# B&R Automation Studio project pneutrunk_plc
Automation Studio 4.9

## Configuration Config1

### Task classes (Cpu.sw)
```
Cyclic#1 (cycle 2000 us, tolerance 2000 us):
  Server <- Source.UDP.Server.prg
  Client <- Source.UDP.Client.prg
  Receiver <- (binary)
  Sender <- (binary)
Cyclic#2 (cycle 12000 us, tolerance 12000 us):
  Receiver1 <- Source.RS485.Receiver.prg
  test_input <- test_input.prg (AdditionalIncludeDirectories=\Logical\MATLAB_includes\R2023a\, BuildOptions=-lm -DMODEL=simulink_2_plc -DNUMST=2 -DNCSTATES=0 -DHAVESTDIO -DRT -DUSE_RTMODEL -DEXT_MODE -DEXTMODE_STATIC -DEXTMODE_STATIC_SIZE=1000000 -DON_TARGET_WAIT_FOR_START=0 -DCLASSIC_INTERFACE=1 -DALLOCATIONFCN=0 -DTID01EQ=1 -DMAT_FILE=0 -DONESTEPFCN=0 -DTERMFCN=1 -DMULTI_INSTANCE_CODE=0 -DINTEGER_CODE=0 -DMT=0 )
Cyclic#3 (cycle 16000 us, tolerance 16000 us):
  Sender1 <- Source.RS485.Sender.prg
  solo_reg <- solo_reg.prg (AdditionalIncludeDirectories=\Logical\MATLAB_includes\R2023a\, BuildOptions=-lm -DMODEL=pneutr2_reg_FF_stiff -DNUMST=1 -DNCSTATES=0 -DHAVESTDIO -DRT -DUSE_RTMODEL -DCLASSIC_INTERFACE=1 -DALLOCATIONFCN=0 -DTID01EQ=0 -DMAT_FILE=0 -DONESTEPFCN=0 -DTERMFCN=1 -DMULTI_INSTANCE_CODE=0 -DINTEGER_CODE=0 -DMT=0 )
Cyclic#4 (cycle 24000 us, tolerance 96000 us):
  Controller <- Source.Controller.prg
  Identifika <- Source.Identifikacia.prg [disabled]
  meranie <- meranie.prg [disabled] (AdditionalIncludeDirectories=\Logical\MATLAB_includes\R2022b\, BuildOptions=-lm -DMODEL=pneutrunkMeranie -DNUMST=1 -DNCSTATES=0 -DHAVESTDIO -DRT -DUSE_RTMODEL -DEXT_MODE -DEXTMODE_STATIC -DEXTMODE_STATIC_SIZE=1000000 -DON_TARGET_WAIT_FOR_START=0 -DCLASSIC_INTERFACE=1 -DALLOCATIONFCN=0 -DTID01EQ=0 -DMAT_FILE=0 -DONESTEPFCN=0 -DTERMFCN=1 -DMULTI_INSTANCE_CODE=0 -DINTEGER_CODE=0 -DMT=0 )
  Testing <- Source.Testing.prg [disabled]
  Program <- Source.Program.prg [disabled]
DataObjects: Acp10sys
Binaries: FWRules, TCData, udbdef, asfw, User, iomap, sysconf, arconfig, ashwd, Role, ashwac, Acp10map, acp10cfg
Libraries: runtime, AsUDP, asstring, standard, sys_lib, brsystem, dvframe, AsTCP, AsArLog, regulatory, asieccon, astime, powerlnk, fileio
```

### Hardware
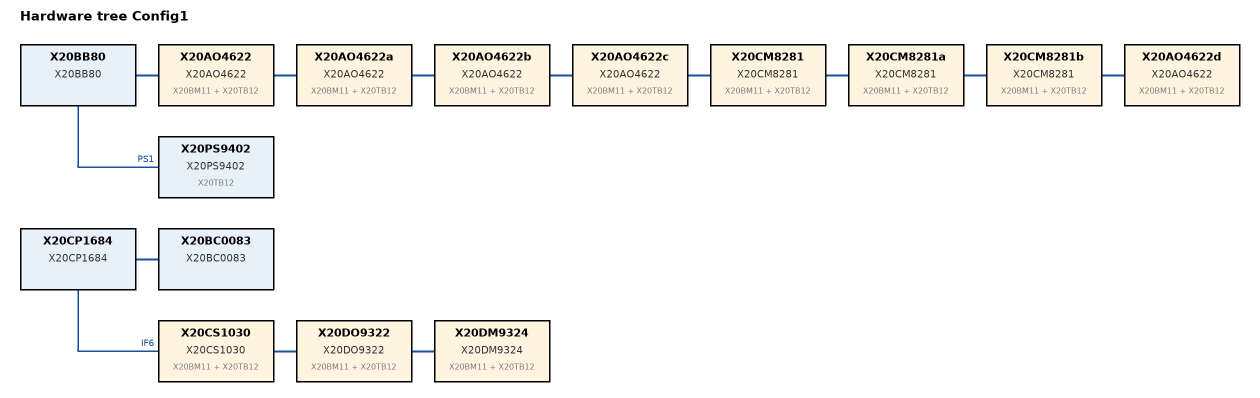
```
X20AO4622 : X20AO4622 v1.3.0.0  [SS1 -> X20TB12a.SS; SL -> X20BM11.SL1]
X20AO4622a : X20AO4622 v1.3.0.0  [SS1 -> X20TB12b.SS; SL -> X20BM11a.SL1]
X20AO4622b : X20AO4622 v1.3.0.0  [SS1 -> X20TB12c.SS; SL -> X20BM11b.SL1]
X20AO4622c : X20AO4622 v1.3.0.0  [SS1 -> X20TB12d.SS; SL -> X20BM11c.SL1]
X20AO4622d : X20AO4622 v1.3.0.0  [SS1 -> X20TB12i.SS; SL -> X20BM11h.SL1]
X20BB80 : X20BB80 v1.1.0.0
X20BC0083 : X20BC0083 v2.14.0.0  [PLK1 -> X20CP1684.IF3 (NodeNumber=1) [Cable Type=PowerlinkCable, Length=10, Version=1.0.0.3]; SL -> X20BB80.SL1]
X20BM11 : X20BM11 v1.1.0.0  [X2X1 -> X20BB80.IF1]
X20BM11a : X20BM11 v1.1.0.0  [X2X1 -> X20BM11.X2X2]
X20BM11b : X20BM11 v1.1.0.0  [X2X1 -> X20BM11a.X2X2]
X20BM11c : X20BM11 v1.1.0.0  [X2X1 -> X20BM11b.X2X2]
X20BM11d : X20BM11 v1.1.0.0  [X2X1 -> X20BM11c.X2X2]
X20BM11e : X20BM11 v1.1.0.0  [X2X1 -> X20BM11d.X2X2]
X20BM11f : X20BM11 v1.1.0.0  [X2X1 -> X20BM11e.X2X2]
X20BM11g : X20BM11 v1.1.0.0  [X2X1 -> X20CP1684.IF6]
X20BM11h : X20BM11 v1.1.0.0  [X2X1 -> X20BM11f.X2X2]
X20BM11i : X20BM11 v1.1.0.0  [X2X1 -> X20BM11g.X2X2]
X20BM11j : X20BM11 v1.1.0.0  [X2X1 -> X20BM11i.X2X2]
X20CM8281 : X20CM8281 v1.4.0.0  [SS1 -> X20TB12e.SS; SL -> X20BM11d.SL1]
X20CM8281a : X20CM8281 v1.4.0.0  [SS1 -> X20TB12f.SS; SL -> X20BM11e.SL1]
X20CM8281b : X20CM8281 v1.4.0.0  [SS1 -> X20TB12g.SS; SL -> X20BM11f.SL1]
X20CP1684 : X20CP1684 v1.5.0.0
  Connector IF2:
    ActivateDevice = 1
    ActivateSnmp = 2
  ConfigurationID = pneutrunk_Config1
  TimerDeviceType = EPLX2X
  TimerDevice = X20CP1684.IF3
  IdleTaskClass = 4
  TaskClassIdleTime = 2000
  Cyclic1Duration = 2000
  Cyclic1Tolerance = 2000
  Cyclic2Duration = 12000
  Cyclic2Tolerance = 12000
  Cyclic3Duration = 16000
  Cyclic3Tolerance = 16000
  Cyclic4Duration = 24000
  Cyclic4Tolerance = 96000
  Cyclic5Duration = 50000
  Cyclic5Tolerance = 50000
  FileDevice1
  FileDeviceName1 = USER
  FileDevicePath1 = USER_PATH
  ActivateDns = 1
  DnsDefaultDomain = br-automation.co.at
  ActivateOpcUa = 1
  OpcUa_Security_AdminRole = Administrators
  OpcUaInformationModels_PV_Version = 1
X20CS1030 : X20CS1030 v1.8.0.0  [SS1 -> X20TB12h.SS; SL -> X20BM11g.SL1]
  Connector IF1:
    Baudrate = 38400
    Parity = N
    DeviceType = RS485
  FunctionModel = StreamCyc1xRS4xx
X20DM9324 : X20DM9324 v1.2.0.0  [SS1 -> X20TB12k.SS; SL -> X20BM11j.SL1]
X20DO9322 : X20DO9322 v1.5.0.0  [SS1 -> X20TB12j.SS; SL -> X20BM11i.SL1]
X20PS9402 : X20PS9402 v1.2.0.0  [SS1 -> X20TB12.SS; PS -> X20BB80.PS1]
X20TB12 : X20TB12 v1.0.0.0
X20TB12a : X20TB12 v1.0.0.0
X20TB12b : X20TB12 v1.0.0.0
X20TB12c : X20TB12 v1.0.0.0
X20TB12d : X20TB12 v1.0.0.0
X20TB12e : X20TB12 v1.0.0.0
X20TB12f : X20TB12 v1.0.0.0
X20TB12g : X20TB12 v1.0.0.0
X20TB12h : X20TB12 v1.0.0.0
X20TB12i : X20TB12 v1.0.0.0
X20TB12j : X20TB12 v1.0.0.0
X20TB12k : X20TB12 v1.0.0.0
```

### IoMap.iom - X20CP1684/IoMap.iom
```iecst
VAR_CONFIG
	::modul.tlak2[5] AT %QW."X20CM8281".AnalogOutput01;
	::modul.tlak3[5] AT %QW."X20CM8281a".AnalogOutput01;
	::modul.tlak1[0] AT %QW."X20AO4622".AnalogOutput01;
	::modul.tlak2[0] AT %QW."X20AO4622".AnalogOutput02;
	::modul.tlak3[0] AT %QW."X20AO4622".AnalogOutput03;
	::modul.tlak1[1] AT %QW."X20AO4622".AnalogOutput04;
	::modul.tlak2[1] AT %QW."X20AO4622a".AnalogOutput01;
	::modul.tlak3[1] AT %QW."X20AO4622a".AnalogOutput02;
	::modul.tlak1[2] AT %QW."X20AO4622a".AnalogOutput03;
	::modul.tlak2[2] AT %QW."X20AO4622a".AnalogOutput04;
	::modul.tlak3[2] AT %QW."X20AO4622b".AnalogOutput01;
	::modul.tlak1[3] AT %QW."X20AO4622b".AnalogOutput02;
	::modul.tlak2[3] AT %QW."X20AO4622b".AnalogOutput03;
	::modul.tlak3[3] AT %QW."X20AO4622b".AnalogOutput04;
	::modul.tlak1[4] AT %QW."X20AO4622c".AnalogOutput01;
	::modul.tlak2[4] AT %QW."X20AO4622c".AnalogOutput02;
	::modul.tlak3[4] AT %QW."X20AO4622c".AnalogOutput03;
	::modul.tlak1[5] AT %QW."X20AO4622c".AnalogOutput04;
	::modul.tlakLinear AT %QW."X20CM8281b".AnalogOutput01;
	::Controller:modull.efektor AT %QX."X20CM8281".DigitalOutput01;
	::modul.tlak2[6] AT %QW."X20AO4622d".AnalogOutput01;
	::modul.tlak3[6] AT %QW."X20AO4622d".AnalogOutput02;
	::modul.tlak1[6] AT %QW."X20AO4622d".AnalogOutput03;
	::zasobnik.ball AT %QX."X20DO9322".DigitalOutput12;
	::zasobnik.ball_piston_sjf AT %QX."X20DO9322".DigitalOutput11;
	::zasobnik.ball_piston AT %QX."X20DO9322".DigitalOutput10;
	::zasobnik.levitovanie AT %QX."X20DO9322".DigitalOutput09;
	::buttons.stropCervenaLED AT %QX."X20DO9322".DigitalOutput08;
	::buttons.startLED AT %QX."X20DO9322".DigitalOutput06;
	::buttons.stopLED AT %QX."X20DO9322".DigitalOutput07;
	::buttons.stropBielaLED AT %QX."X20DO9322".DigitalOutput05;
	::buttons.startButton AT %IX."X20DM9324".DigitalInput01;
	::buttons.stop AT %IX."X20DM9324".DigitalInput02;
	::buttons.centralStop AT %IX."X20DM9324".DigitalInput04;
END_VAR
```

## Logical view

### Global.typ - Global data types
```iecst
TYPE
	tlacidla : 	STRUCT
		start : BOOL;
		ros : BOOL;
		stopLED : BOOL;
		stop : BOOL;
		startLED : BOOL;
		startButton : BOOL;
		centralStop : BOOL;
		stropBielaLED : BOOL;
		stropCervenaLED : BOOL;
		klucik : BOOL;
	END_STRUCT;
	automatic : 	STRUCT
		y_desired : ARRAY[0..6]OF INT := [7(0)];
		x_desired : ARRAY[0..6]OF INT := [7(0)];
		linear : INT;
		ball_up : BOOL;
		casovac : BOOL;
		effector : BOOL;
		casovac_uchopenie : BOOL;
		ball_piston : BOOL;
		novyCyklus : TIME := T#1s;
		novyCyklusStart : BOOL;
		trajectoryStart2 : BOOL;
		trajectoryTime2 : TIME := T#6s;
		automatic : BOOL;
		holdPosition : BOOL;
		cas : INT;
		box : INT;
		step_color : INT;
		popcorn : BOOL;
		testFarba : INT;
		loptickyVzasobniku : BOOL := TRUE;
		x_desired_previous : ARRAY[0..6]OF INT;
		y_desired_previous : ARRAY[0..6]OF INT;
		I_konstanta : ARRAY[0..6]OF INT;
		levitacia : BOOL;
	END_STRUCT;
	podavac : 	STRUCT
		levitovanie : BOOL;
		ball_piston_sjf : BOOL;
		ball : BOOL;
		ball_piston : BOOL;
	END_STRUCT;
	identifikacia : 	STRUCT
		p3 : REAL;
		p2 : REAL;
		p1 : REAL;
		vzorka : USINT;
		uhol2 : ARRAY[0..9]OF INT;
		uhol2Priemer : INT;
		uhol1Priemer : INT;
		uhol1 : ARRAY[0..9]OF INT;
		uhol2Stabilny : BOOL;
		uhol1Stabilny : BOOL;
		uhol2Ref : INT;
		uhol1Ref : INT;
		krok : USINT;
		p2Mem : REAL;
		p1Mem : REAL;
		tonStart : BOOL;
		pocetOverenie : USINT := 10;
		spustit : BOOL;
		p3Koniec : BOOL;
		p2Koniec : BOOL;
		p1Koniec : BOOL;
		p3Mem : REAL;
		results : INT;
		switchs : BOOL;
		inkrement : REAL;
		hornyTlak : REAL;
	END_STRUCT;
	packetRS485 : 	STRUCT
		packet : ARRAY[0..9]OF BYTE;
		sendPacketLED : ARRAY[0..5]OF BYTE;
		sendPacketSnimace : ARRAY[0..5]OF BYTE;
		sendPacketFinal : ARRAY[0..5]OF BYTE;
		id : USINT;
	END_STRUCT;
	packetUDP : 	STRUCT
		qLength : INT;
		c : INT;
		q : INT;
		qFull : STRING[80];
		comma : INT;
		qString : ARRAY[0..14]OF STRING[6];
		qDesired : ARRAY[0..14]OF REAL;
		color : INT;
		step : INT;
	END_STRUCT;
	tlaky : 	STRUCT
		tlak3 : USINT;
		tlak2 : USINT;
		tlak1 : USINT;
	END_STRUCT;
	moduly : 	STRUCT
		uhol2 : ARRAY[0..6]OF INT := [7(0)];
		uhol1 : ARRAY[0..6]OF INT := [7(0)];
		koncak : ARRAY[0..6]OF BOOL;
		led : ARRAY[0..6]OF BOOL;
		uholINT2 : INT;
		uholINT1 : INT;
		tlak1 : ARRAY[0..6]OF INT;
		tlak2 : ARRAY[0..6]OF INT;
		tlak3 : ARRAY[0..6]OF INT;
		tlakLinear : INT;
		uhol_XminusRef : ARRAY[0..6]OF REAL; (*uhol ktory posiela PLC do PC po odpocitani odchylky naklonenia realneho robota*)
		uhol_YminusRef : ARRAY[0..6]OF REAL; (*uhol ktory posiela PLC do PC po odpocitani odchylky naklonenia realneho robota*)
		linearReal : REAL;
		naraz : ARRAY[0..7]OF BOOL;
		narazAktivny : BOOL;
	END_STRUCT;
END_TYPE
```

### Global.var - Global variables
```iecst
VAR
	hranica_upravy_traj : REAL := 2;
	Yellow_tab_ID7 : REAL;
	zasobnik : podavac;
	Yellow_tab_ID6 : REAL;
	I_ON : BOOL;
	Yellow_tab_ID5 : REAL;
	step : INT;
	Yellow_tab_ID4 : REAL;
	Yellow_tab_ID3 : REAL;
	Yellow_tab_ID2 : REAL;
	automatika : automatic;
	Yellow_tab_ID1 : REAL;
	u2 : INT;
	u1 : INT;
	stiffness_ff : REAL;
	result : INT;
	RESET_ID7 : REAL;
	RESET_ID6 : REAL;
	RESET_ID5 : REAL;
	RESET_ID4 : REAL;
	RESET_ID3 : REAL;
	RESET_ID2 : REAL;
	RESET_ID1 : REAL;
	ref_linearny_posun : REAL;
	ref_alfa_y_ID7 : REAL;
	ref_alfa_y_ID6 : REAL;
	ref_alfa_y_ID5 : REAL;
	ref_alfa_y_ID4 : REAL;
	ref_alfa_y_ID3 : REAL;
	ref_alfa_y_ID2 : REAL;
	ref_alfa_y_ID1 : REAL;
	ref_alfa_x_ID7 : REAL;
	ref_alfa_x_ID6 : REAL;
	ref_alfa_x_ID5 : REAL;
	ref_alfa_x_ID4 : REAL;
	ref_alfa_x_ID3 : REAL;
	ref_alfa_x_ID2 : REAL;
	ref_alfa_x_ID1 : REAL;
	q_real : ARRAY[0..12] OF REAL := [0.55,12.58,12.23,7.85,1.23,15.36,17.85,12.05,3.85,3.6,-12.52,10.65,31.28];
	q_desired : ARRAY[0..12] OF REAL;
	pripustna_odchylka_naklonenia : REAL := 0.25;
	poradie_ID7 : REAL;
	poradie_ID6 : REAL;
	poradie_ID5 : REAL;
	poradie_ID4 : REAL;
	poradie_ID3 : REAL;
	poradie_ID2 : REAL;
	poradie_ID1 : REAL;
	packetPos : packetUDP;
	packet485 : packetRS485;
	p3 : REAL;
	p2 : REAL;
	p1 : REAL;
	modul : moduly;
	meranie : identifikacia;
	lin_pressure : REAL;
	I_konstanta_ID7 : REAL;
	I_konstanta_ID6 : REAL;
	I_konstanta_ID5 : REAL;
	I_konstanta_ID4 : REAL;
	I_konstanta_ID3 : REAL;
	I_konstanta_ID2 : REAL;
	cos_test_hodnota2 : REAL;
	cos_test_hodnota1 : REAL;
	I_konstanta_ID1 : REAL;
	Green_tab_ID7 : REAL;
	Green_tab_ID6 : REAL;
	trajectoryStart : BOOL;
	Green_tab_ID5 : REAL;
	Green_tab_ID4 : REAL;
	uhly : experimentyUhly;
	Green_tab_ID3 : REAL;
	Green_tab_ID2 : REAL;
	Green_tab_ID1 : REAL;
	step_color : INT;
	global_step_udp : INT;
	global_step : INT;
	datagramLength : INT;
	centralStop : BOOL;
	cas_trajektorie : REAL := 100;
	Blue_tab_ID7 : REAL;
	Blue_tab_ID6 : REAL;
	Blue_tab_ID5 : REAL;
	buttons : tlacidla;
	Blue_tab_ID4 : REAL;
	Blue_tab_ID3 : REAL;
	Blue_tab_ID2 : REAL;
	Blue_tab_ID1 : REAL;
	act_alfa_y_ID7 : REAL;
	act_alfa_y_ID6 : REAL;
	act_alfa_y_ID5 : REAL;
	step_repeatability : INT;
	act_alfa_y_ID4 : REAL;
	act_alfa_y_ID3 : REAL;
	act_alfa_y_ID2 : REAL;
	act_alfa_y_ID1 : REAL;
	act_alfa_x_ID7 : REAL;
	act_alfa_x_ID6 : REAL;
	act_alfa_x_ID5 : REAL;
	act_alfa_x_ID4 : REAL;
	act_alfa_x_ID3 : REAL;
	act_alfa_x_ID2 : REAL;
	act_alfa_x_ID1 : REAL;
END_VAR
```

### Package Logical/Libraries - Global libraries

### Program Logical/Libraries/regulatory

#### multiword_types.h
```c
/*
 * multiword_types.h
 *
 * Academic License - for use in teaching, academic research, and meeting
 * course requirements at degree granting institutions only.  Not for
 * government, commercial, or other organizational use.
 *
 * Code generation for model "reg_FF_PI_pl_regr_stiff".
 *
 * Model version              : 1.154
 * Simulink Coder version : 9.6 (R2021b) 14-May-2021
 * C source code generated on : Mon Jun 26 09:10:26 2023
 *
 * Target selection: bur_grt.tlc
 * Note: GRT includes extra infrastructure and instrumentation for prototyping
 * Embedded hardware selection: Intel->x86/Pentium
 * Code generation objectives: Unspecified
 * Validation result: Not run
 */

#ifndef MULTIWORD_TYPES_H
#define MULTIWORD_TYPES_H
#include "rtwtypes.h"

/*
 * MultiWord supporting definitions
 */
typedef long int long_T;

/*
 * MultiWord types
 */
typedef struct {
  uint32_T chunks[2];
} int64m_T;

typedef struct {
  int64m_T re;
  int64m_T im;
} cint64m_T;

typedef struct {
  uint32_T chunks[2];
} uint64m_T;

typedef struct {
  uint64m_T re;
  uint64m_T im;
} cuint64m_T;

typedef struct {
  uint32_T chunks[3];
} int96m_T;

typedef struct {
  int96m_T re;
  int96m_T im;
} cint96m_T;

typedef struct {
  uint32_T chunks[3];
} uint96m_T;

typedef struct {
  uint96m_T re;
  uint96m_T im;
} cuint96m_T;

typedef struct {
  uint32_T chunks[4];
} int128m_T;

typedef struct {
  int128m_T re;
  int128m_T im;
} cint128m_T;

typedef struct {
  uint32_T chunks[4];
} uint128m_T;

typedef struct {
  uint128m_T re;
  uint128m_T im;
} cuint128m_T;

typedef struct {
  uint32_T chunks[5];
} int160m_T;

typedef struct {
  int160m_T re;
  int160m_T im;
} cint160m_T;

typedef struct {
  uint32_T chunks[5];
} uint160m_T;

typedef struct {
  uint160m_T re;
  uint160m_T im;
} cuint160m_T;

typedef struct {
  uint32_T chunks[6];
} int192m_T;

typedef struct {
  int192m_T re;
  int192m_T im;
} cint192m_T;

typedef struct {
  uint32_T chunks[6];
} uint192m_T;

typedef struct {
  uint192m_T re;
  uint192m_T im;
} cuint192m_T;

typedef struct {
  uint32_T chunks[7];
} int224m_T;

typedef struct {
  int224m_T re;
  int224m_T im;
} cint224m_T;

typedef struct {
  uint32_T chunks[7];
} uint224m_T;

typedef struct {
  uint224m_T re;
  uint224m_T im;
} cuint224m_T;

typedef struct {
  uint32_T chunks[8];
} int256m_T;

typedef struct {
  int256m_T re;
  int256m_T im;
} cint256m_T;

typedef struct {
  uint32_T chunks[8];
} uint256m_T;

typedef struct {
  uint256m_T re;
  uint256m_T im;
} cuint256m_T;

typedef struct {
  uint32_T chunks[9];
} int288m_T;

typedef struct {
  int288m_T re;
  int288m_T im;
} cint288m_T;

typedef struct {
  uint32_T chunks[9];
} uint288m_T;

typedef struct {
  uint288m_T re;
  uint288m_T im;
} cuint288m_T;

typedef struct {
  uint32_T chunks[10];
} int320m_T;

typedef struct {
  int320m_T re;
  int320m_T im;
} cint320m_T;

typedef struct {
  uint32_T chunks[10];
} uint320m_T;

typedef struct {
  uint320m_T re;
  uint320m_T im;
} cuint320m_T;

typedef struct {
  uint32_T chunks[11];
} int352m_T;

typedef struct {
  int352m_T re;
  int352m_T im;
} cint352m_T;

typedef struct {
  uint32_T chunks[11];
} uint352m_T;

typedef struct {
  uint352m_T re;
  uint352m_T im;
} cuint352m_T;

typedef struct {
  uint32_T chunks[12];
} int384m_T;

typedef struct {
  int384m_T re;
  int384m_T im;
} cint384m_T;

typedef struct {
  uint32_T chunks[12];
} uint384m_T;

typedef struct {
  uint384m_T re;
  uint384m_T im;
} cuint384m_T;

typedef struct {
  uint32_T chunks[13];
} int416m_T;

typedef struct {
  int416m_T re;
  int416m_T im;
} cint416m_T;

typedef struct {
  uint32_T chunks[13];
} uint416m_T;

typedef struct {
  uint416m_T re;
  uint416m_T im;
} cuint416m_T;

typedef struct {
  uint32_T chunks[14];
} int448m_T;

typedef struct {
  int448m_T re;
  int448m_T im;
} cint448m_T;

typedef struct {
  uint32_T chunks[14];
} uint448m_T;

typedef struct {
  uint448m_T re;
  uint448m_T im;
} cuint448m_T;

typedef struct {
  uint32_T chunks[15];
} int480m_T;

typedef struct {
  int480m_T re;
  int480m_T im;
} cint480m_T;

typedef struct {
  uint32_T chunks[15];
} uint480m_T;

typedef struct {
  uint480m_T re;
  uint480m_T im;
} cuint480m_T;

typedef struct {
  uint32_T chunks[16];
} int512m_T;

typedef struct {
  int512m_T re;
  int512m_T im;
} cint512m_T;

typedef struct {
  uint32_T chunks[16];
} uint512m_T;

typedef struct {
  uint512m_T re;
  uint512m_T im;
} cuint512m_T;

typedef struct {
  uint32_T chunks[17];
} int544m_T;

typedef struct {
  int544m_T re;
  int544m_T im;
} cint544m_T;

typedef struct {
  uint32_T chunks[17];
} uint544m_T;

typedef struct {
  uint544m_T re;
  uint544m_T im;
} cuint544m_T;

typedef struct {
  uint32_T chunks[18];
} int576m_T;

typedef struct {
  int576m_T re;
  int576m_T im;
} cint576m_T;

typedef struct {
  uint32_T chunks[18];
} uint576m_T;

typedef struct {
  uint576m_T re;
  uint576m_T im;
} cuint576m_T;

typedef struct {
  uint32_T chunks[19];
} int608m_T;

typedef struct {
  int608m_T re;
  int608m_T im;
} cint608m_T;

typedef struct {
  uint32_T chunks[19];
} uint608m_T;

typedef struct {
  uint608m_T re;
  uint608m_T im;
} cuint608m_T;

typedef struct {
  uint32_T chunks[20];
} int640m_T;

typedef struct {
  int640m_T re;
  int640m_T im;
} cint640m_T;

typedef struct {
  uint32_T chunks[20];
} uint640m_T;

typedef struct {
  uint640m_T re;
  uint640m_T im;
} cuint640m_T;

typedef struct {
  uint32_T chunks[21];
} int672m_T;

typedef struct {
  int672m_T re;
  int672m_T im;
} cint672m_T;

typedef struct {
  uint32_T chunks[21];
} uint672m_T;

typedef struct {
  uint672m_T re;
  uint672m_T im;
} cuint672m_T;

typedef struct {
  uint32_T chunks[22];
} int704m_T;

typedef struct {
  int704m_T re;
  int704m_T im;
} cint704m_T;

typedef struct {
  uint32_T chunks[22];
} uint704m_T;

typedef struct {
  uint704m_T re;
  uint704m_T im;
} cuint704m_T;

typedef struct {
  uint32_T chunks[23];
} int736m_T;

typedef struct {
  int736m_T re;
  int736m_T im;
} cint736m_T;

typedef struct {
  uint32_T chunks[23];
} uint736m_T;

typedef struct {
  uint736m_T re;
  uint736m_T im;
} cuint736m_T;

typedef struct {
  uint32_T chunks[24];
} int768m_T;

typedef struct {
  int768m_T re;
  int768m_T im;
} cint768m_T;

typedef struct {
  uint32_T chunks[24];
} uint768m_T;

typedef struct {
  uint768m_T re;
  uint768m_T im;
} cuint768m_T;

typedef struct {
  uint32_T chunks[25];
} int800m_T;

typedef struct {
  int800m_T re;
  int800m_T im;
} cint800m_T;

typedef struct {
  uint32_T chunks[25];
} uint800m_T;

typedef struct {
  uint800m_T re;
  uint800m_T im;
} cuint800m_T;

typedef struct {
  uint32_T chunks[26];
} int832m_T;

typedef struct {
  int832m_T re;
  int832m_T im;
} cint832m_T;

typedef struct {
  uint32_T chunks[26];
} uint832m_T;

typedef struct {
  uint832m_T re;
  uint832m_T im;
} cuint832m_T;

typedef struct {
  uint32_T chunks[27];
} int864m_T;

typedef struct {
  int864m_T re;
  int864m_T im;
} cint864m_T;

typedef struct {
  uint32_T chunks[27];
} uint864m_T;

typedef struct {
  uint864m_T re;
  uint864m_T im;
} cuint864m_T;

typedef struct {
  uint32_T chunks[28];
} int896m_T;

typedef struct {
  int896m_T re;
  int896m_T im;
} cint896m_T;

typedef struct {
  uint32_T chunks[28];
} uint896m_T;

typedef struct {
  uint896m_T re;
  uint896m_T im;
} cuint896m_T;

typedef struct {
  uint32_T chunks[29];
} int928m_T;

typedef struct {
  int928m_T re;
  int928m_T im;
} cint928m_T;

typedef struct {
  uint32_T chunks[29];
} uint928m_T;

typedef struct {
  uint928m_T re;
  uint928m_T im;
} cuint928m_T;

typedef struct {
  uint32_T chunks[30];
} int960m_T;

typedef struct {
  int960m_T re;
  int960m_T im;
} cint960m_T;

typedef struct {
  uint32_T chunks[30];
} uint960m_T;

typedef struct {
  uint960m_T re;
  uint960m_T im;
} cuint960m_T;

typedef struct {
  uint32_T chunks[31];
} int992m_T;

typedef struct {
  int992m_T re;
  int992m_T im;
} cint992m_T;

typedef struct {
  uint32_T chunks[31];
} uint992m_T;

typedef struct {
  uint992m_T re;
  uint992m_T im;
} cuint992m_T;

typedef struct {
  uint32_T chunks[32];
} int1024m_T;

typedef struct {
  int1024m_T re;
  int1024m_T im;
} cint1024m_T;

typedef struct {
  uint32_T chunks[32];
} uint1024m_T;

typedef struct {
  uint1024m_T re;
  uint1024m_T im;
} cuint1024m_T;

typedef struct {
  uint32_T chunks[33];
} int1056m_T;

typedef struct {
  int1056m_T re;
  int1056m_T im;
} cint1056m_T;

typedef struct {
  uint32_T chunks[33];
} uint1056m_T;

typedef struct {
  uint1056m_T re;
  uint1056m_T im;
} cuint1056m_T;

typedef struct {
  uint32_T chunks[34];
} int1088m_T;

typedef struct {
  int1088m_T re;
  int1088m_T im;
} cint1088m_T;

typedef struct {
  uint32_T chunks[34];
} uint1088m_T;

typedef struct {
  uint1088m_T re;
  uint1088m_T im;
} cuint1088m_T;

typedef struct {
  uint32_T chunks[35];
} int1120m_T;

typedef struct {
  int1120m_T re;
  int1120m_T im;
} cint1120m_T;

typedef struct {
  uint32_T chunks[35];
} uint1120m_T;

typedef struct {
  uint1120m_T re;
  uint1120m_T im;
} cuint1120m_T;

typedef struct {
  uint32_T chunks[36];
} int1152m_T;

typedef struct {
  int1152m_T re;
  int1152m_T im;
} cint1152m_T;

typedef struct {
  uint32_T chunks[36];
} uint1152m_T;

typedef struct {
  uint1152m_T re;
  uint1152m_T im;
} cuint1152m_T;

typedef struct {
  uint32_T chunks[37];
} int1184m_T;

typedef struct {
  int1184m_T re;
  int1184m_T im;
} cint1184m_T;

typedef struct {
  uint32_T chunks[37];
} uint1184m_T;

typedef struct {
  uint1184m_T re;
  uint1184m_T im;
} cuint1184m_T;

typedef struct {
  uint32_T chunks[38];
} int1216m_T;

typedef struct {
  int1216m_T re;
  int1216m_T im;
} cint1216m_T;

typedef struct {
  uint32_T chunks[38];
} uint1216m_T;

typedef struct {
  uint1216m_T re;
  uint1216m_T im;
} cuint1216m_T;

typedef struct {
  uint32_T chunks[39];
} int1248m_T;

typedef struct {
  int1248m_T re;
  int1248m_T im;
} cint1248m_T;

typedef struct {
  uint32_T chunks[39];
} uint1248m_T;

typedef struct {
  uint1248m_T re;
  uint1248m_T im;
} cuint1248m_T;

typedef struct {
  uint32_T chunks[40];
} int1280m_T;

typedef struct {
  int1280m_T re;
  int1280m_T im;
} cint1280m_T;

typedef struct {
  uint32_T chunks[40];
} uint1280m_T;

typedef struct {
  uint1280m_T re;
  uint1280m_T im;
} cuint1280m_T;

typedef struct {
  uint32_T chunks[41];
} int1312m_T;

typedef struct {
  int1312m_T re;
  int1312m_T im;
} cint1312m_T;

typedef struct {
  uint32_T chunks[41];
} uint1312m_T;

typedef struct {
  uint1312m_T re;
  uint1312m_T im;
} cuint1312m_T;

typedef struct {
  uint32_T chunks[42];
} int1344m_T;

typedef struct {
  int1344m_T re;
  int1344m_T im;
} cint1344m_T;

typedef struct {
  uint32_T chunks[42];
} uint1344m_T;

typedef struct {
  uint1344m_T re;
  uint1344m_T im;
} cuint1344m_T;

typedef struct {
  uint32_T chunks[43];
} int1376m_T;

typedef struct {
  int1376m_T re;
  int1376m_T im;
} cint1376m_T;

typedef struct {
  uint32_T chunks[43];
} uint1376m_T;

typedef struct {
  uint1376m_T re;
  uint1376m_T im;
} cuint1376m_T;

typedef struct {
  uint32_T chunks[44];
} int1408m_T;

typedef struct {
  int1408m_T re;
  int1408m_T im;
} cint1408m_T;

typedef struct {
  uint32_T chunks[44];
} uint1408m_T;

typedef struct {
  uint1408m_T re;
  uint1408m_T im;
} cuint1408m_T;

typedef struct {
  uint32_T chunks[45];
} int1440m_T;

typedef struct {
  int1440m_T re;
  int1440m_T im;
} cint1440m_T;

typedef struct {
  uint32_T chunks[45];
} uint1440m_T;

typedef struct {
  uint1440m_T re;
  uint1440m_T im;
} cuint1440m_T;

typedef struct {
  uint32_T chunks[46];
} int1472m_T;

typedef struct {
  int1472m_T re;
  int1472m_T im;
} cint1472m_T;

typedef struct {
  uint32_T chunks[46];
} uint1472m_T;

typedef struct {
  uint1472m_T re;
  uint1472m_T im;
} cuint1472m_T;

typedef struct {
  uint32_T chunks[47];
} int1504m_T;

typedef struct {
  int1504m_T re;
  int1504m_T im;
} cint1504m_T;

typedef struct {
  uint32_T chunks[47];
} uint1504m_T;

typedef struct {
  uint1504m_T re;
  uint1504m_T im;
} cuint1504m_T;

typedef struct {
  uint32_T chunks[48];
} int1536m_T;

typedef struct {
  int1536m_T re;
  int1536m_T im;
} cint1536m_T;

typedef struct {
  uint32_T chunks[48];
} uint1536m_T;

typedef struct {
  uint1536m_T re;
  uint1536m_T im;
} cuint1536m_T;

typedef struct {
  uint32_T chunks[49];
} int1568m_T;

typedef struct {
  int1568m_T re;
  int1568m_T im;
} cint1568m_T;

typedef struct {
  uint32_T chunks[49];
} uint1568m_T;

typedef struct {
  uint1568m_T re;
  uint1568m_T im;
} cuint1568m_T;

typedef struct {
  uint32_T chunks[50];
} int1600m_T;

typedef struct {
  int1600m_T re;
  int1600m_T im;
} cint1600m_T;

typedef struct {
  uint32_T chunks[50];
} uint1600m_T;

typedef struct {
  uint1600m_T re;
  uint1600m_T im;
} cuint1600m_T;

typedef struct {
  uint32_T chunks[51];
} int1632m_T;

typedef struct {
  int1632m_T re;
  int1632m_T im;
} cint1632m_T;

typedef struct {
  uint32_T chunks[51];
} uint1632m_T;

typedef struct {
  uint1632m_T re;
  uint1632m_T im;
} cuint1632m_T;

typedef struct {
  uint32_T chunks[52];
} int1664m_T;

typedef struct {
  int1664m_T re;
  int1664m_T im;
} cint1664m_T;

typedef struct {
  uint32_T chunks[52];
} uint1664m_T;

typedef struct {
  uint1664m_T re;
  uint1664m_T im;
} cuint1664m_T;

typedef struct {
  uint32_T chunks[53];
} int1696m_T;

typedef struct {
  int1696m_T re;
  int1696m_T im;
} cint1696m_T;

typedef struct {
  uint32_T chunks[53];
} uint1696m_T;

typedef struct {
  uint1696m_T re;
  uint1696m_T im;
} cuint1696m_T;

typedef struct {
  uint32_T chunks[54];
} int1728m_T;

typedef struct {
  int1728m_T re;
  int1728m_T im;
} cint1728m_T;

typedef struct {
  uint32_T chunks[54];
} uint1728m_T;

typedef struct {
  uint1728m_T re;
  uint1728m_T im;
} cuint1728m_T;

typedef struct {
  uint32_T chunks[55];
} int1760m_T;

typedef struct {
  int1760m_T re;
  int1760m_T im;
} cint1760m_T;

typedef struct {
  uint32_T chunks[55];
} uint1760m_T;

typedef struct {
  uint1760m_T re;
  uint1760m_T im;
} cuint1760m_T;

typedef struct {
  uint32_T chunks[56];
} int1792m_T;

typedef struct {
  int1792m_T re;
  int1792m_T im;
} cint1792m_T;

typedef struct {
  uint32_T chunks[56];
} uint1792m_T;

typedef struct {
  uint1792m_T re;
  uint1792m_T im;
} cuint1792m_T;

typedef struct {
  uint32_T chunks[57];
} int1824m_T;

typedef struct {
  int1824m_T re;
  int1824m_T im;
} cint1824m_T;

typedef struct {
  uint32_T chunks[57];
} uint1824m_T;

typedef struct {
  uint1824m_T re;
  uint1824m_T im;
} cuint1824m_T;

typedef struct {
  uint32_T chunks[58];
} int1856m_T;

typedef struct {
  int1856m_T re;
  int1856m_T im;
} cint1856m_T;

typedef struct {
  uint32_T chunks[58];
} uint1856m_T;

typedef struct {
  uint1856m_T re;
  uint1856m_T im;
} cuint1856m_T;

typedef struct {
  uint32_T chunks[59];
} int1888m_T;

typedef struct {
  int1888m_T re;
  int1888m_T im;
} cint1888m_T;

typedef struct {
  uint32_T chunks[59];
} uint1888m_T;

typedef struct {
  uint1888m_T re;
  uint1888m_T im;
} cuint1888m_T;

typedef struct {
  uint32_T chunks[60];
} int1920m_T;

typedef struct {
  int1920m_T re;
  int1920m_T im;
} cint1920m_T;

typedef struct {
  uint32_T chunks[60];
} uint1920m_T;

typedef struct {
  uint1920m_T re;
  uint1920m_T im;
} cuint1920m_T;

typedef struct {
  uint32_T chunks[61];
} int1952m_T;

typedef struct {
  int1952m_T re;
  int1952m_T im;
} cint1952m_T;

typedef struct {
  uint32_T chunks[61];
} uint1952m_T;

typedef struct {
  uint1952m_T re;
  uint1952m_T im;
} cuint1952m_T;

typedef struct {
  uint32_T chunks[62];
} int1984m_T;

typedef struct {
  int1984m_T re;
  int1984m_T im;
} cint1984m_T;

typedef struct {
  uint32_T chunks[62];
} uint1984m_T;

typedef struct {
  uint1984m_T re;
  uint1984m_T im;
} cuint1984m_T;

typedef struct {
  uint32_T chunks[63];
} int2016m_T;

typedef struct {
  int2016m_T re;
  int2016m_T im;
} cint2016m_T;

typedef struct {
  uint32_T chunks[63];
} uint2016m_T;

typedef struct {
  uint2016m_T re;
  uint2016m_T im;
} cuint2016m_T;

typedef struct {
  uint32_T chunks[64];
} int2048m_T;

typedef struct {
  int2048m_T re;
  int2048m_T im;
} cint2048m_T;

typedef struct {
  uint32_T chunks[64];
} uint2048m_T;

typedef struct {
  uint2048m_T re;
  uint2048m_T im;
} cuint2048m_T;

#endif                                 /* MULTIWORD_TYPES_H */
```

#### PID_co_private.h
```c
/*
 * PID_co_private.h
 *
 * Academic License - for use in teaching, academic research, and meeting
 * course requirements at degree granting institutions only.  Not for
 * government, commercial, or other organizational use.
 *
 * Code generation for model "PID_co".
 *
 * Model version              : 1.9
 * Simulink Coder version : 9.6 (R2021b) 14-May-2021
 * C source code generated on : Mon Sep 26 14:43:58 2022
 *
 * Target selection: bur_grt.tlc
 * Note: GRT includes extra infrastructure and instrumentation for prototyping
 * Embedded hardware selection: Intel->x86/Pentium
 * Code generation objectives: Unspecified
 * Validation result: Not run
 */

#ifndef RTW_HEADER_PID_co_private_h_
#define RTW_HEADER_PID_co_private_h_
#include "rtwtypes.h"
#include "multiword_types.h"
#if !defined(rt_VALIDATE_MEMORY)
#define rt_VALIDATE_MEMORY(S, ptr)     if(!(ptr)) {\
 rtmSetErrorStatus(PID_co_M, RT_MEMORY_ALLOCATION_ERROR);\
 }
#endif

#if !defined(rt_FREE)
#if !defined(_WIN32)
#define rt_FREE(ptr)                   if((ptr) != (NULL)) {\
 free((ptr));\
 (ptr) = (NULL);\
 }
#else

/* Visual and other windows compilers declare free without const */
#define rt_FREE(ptr)                   if((ptr) != (NULL)) {\
 free((void *)(ptr));\
 (ptr) = (NULL);\
 }
#endif
#endif
#endif                                 /* RTW_HEADER_PID_co_private_h_ */
```

#### PID_co_types.h
```c
/*
 * PID_co_types.h
 *
 * Academic License - for use in teaching, academic research, and meeting
 * course requirements at degree granting institutions only.  Not for
 * government, commercial, or other organizational use.
 *
 * Code generation for model "PID_co".
 *
 * Model version              : 1.9
 * Simulink Coder version : 9.6 (R2021b) 14-May-2021
 * C source code generated on : Mon Sep 26 14:43:58 2022
 *
 * Target selection: bur_grt.tlc
 * Note: GRT includes extra infrastructure and instrumentation for prototyping
 * Embedded hardware selection: Intel->x86/Pentium
 * Code generation objectives: Unspecified
 * Validation result: Not run
 */

#ifndef RTW_HEADER_PID_co_types_h_
#define RTW_HEADER_PID_co_types_h_

/* Model Code Variants */

/* Forward declaration for rtModel */

#endif                                 /* RTW_HEADER_PID_co_types_h_ */
```

#### reg_FF_PI_pl_regr_stiff_private.h
```c
/*
 * reg_FF_PI_pl_regr_stiff_private.h
 *
 * Academic License - for use in teaching, academic research, and meeting
 * course requirements at degree granting institutions only.  Not for
 * government, commercial, or other organizational use.
 *
 * Code generation for model "reg_FF_PI_pl_regr_stiff".
 *
 * Model version              : 1.154
 * Simulink Coder version : 9.6 (R2021b) 14-May-2021
 * C source code generated on : Mon Jun 26 09:10:26 2023
 *
 * Target selection: bur_grt.tlc
 * Note: GRT includes extra infrastructure and instrumentation for prototyping
 * Embedded hardware selection: Intel->x86/Pentium
 * Code generation objectives: Unspecified
 * Validation result: Not run
 */

#ifndef RTW_HEADER_reg_FF_PI_pl_regr_stiff_private_h_
#define RTW_HEADER_reg_FF_PI_pl_regr_stiff_private_h_
#include "rtwtypes.h"
#include "multiword_types.h"
#if !defined(rt_VALIDATE_MEMORY)
#define rt_VALIDATE_MEMORY(S, ptr)     if(!(ptr)) {\
 rtmSetErrorStatus(reg_FF_PI_pl_regr_stiff_M, RT_MEMORY_ALLOCATION_ERROR);\
 }
#endif

#if !defined(rt_FREE)
#if !defined(_WIN32)
#define rt_FREE(ptr)                   if((ptr) != (NULL)) {\
 free((ptr));\
 (ptr) = (NULL);\
 }
#else

/* Visual and other windows compilers declare free without const */
#define rt_FREE(ptr)                   if((ptr) != (NULL)) {\
 free((void *)(ptr));\
 (ptr) = (NULL);\
 }
#endif
#endif
#endif                       /* RTW_HEADER_reg_FF_PI_pl_regr_stiff_private_h_ */
```

#### regulator_nelin_P_types.h
```c
/*
 * regulator_nelin_P_types.h
 *
 * Academic License - for use in teaching, academic research, and meeting
 * course requirements at degree granting institutions only.  Not for
 * government, commercial, or other organizational use.
 *
 * Code generation for model "regulator_nelin_P".
 *
 * Model version              : 1.10
 * Simulink Coder version : 9.6 (R2021b) 14-May-2021
 * C source code generated on : Fri Jul 29 10:48:17 2022
 *
 * Target selection: bur_grt.tlc
 * Note: GRT includes extra infrastructure and instrumentation for prototyping
 * Embedded hardware selection: Intel->x86/Pentium
 * Code generation objectives: Unspecified
 * Validation result: Not run
 */

#ifndef RTW_HEADER_regulator_nelin_P_types_h_
#define RTW_HEADER_regulator_nelin_P_types_h_

/* Model Code Variants */

/* Forward declaration for rtModel */

#endif                               /* RTW_HEADER_regulator_nelin_P_types_h_ */
```

#### rt_defines.h
```c
/*
 * rt_defines.h
 *
 * Academic License - for use in teaching, academic research, and meeting
 * course requirements at degree granting institutions only.  Not for
 * government, commercial, or other organizational use.
 *
 * Code generation for model "regulator_nelin_P".
 *
 * Model version              : 1.10
 * Simulink Coder version : 9.6 (R2021b) 14-May-2021
 * C source code generated on : Fri Jul 29 10:48:17 2022
 *
 * Target selection: bur_grt.tlc
 * Note: GRT includes extra infrastructure and instrumentation for prototyping
 * Embedded hardware selection: Intel->x86/Pentium
 * Code generation objectives: Unspecified
 * Validation result: Not run
 */

#ifndef RTW_HEADER_rt_defines_h_
#define RTW_HEADER_rt_defines_h_

/*===========*
 * Constants *
 *===========*/
#define RT_PI                          3.14159265358979323846
#define RT_PIF                         3.1415927F
#define RT_LN_10                       2.30258509299404568402
#define RT_LN_10F                      2.3025851F
#define RT_LOG10E                      0.43429448190325182765
#define RT_LOG10EF                     0.43429449F
#define RT_E                           2.7182818284590452354
#define RT_EF                          2.7182817F

/*
 * UNUSED_PARAMETER(x)
 *   Used to specify that a function parameter (argument) is required but not
 *   accessed by the function body.
 */
#ifndef UNUSED_PARAMETER
#if defined(__LCC__)
#define UNUSED_PARAMETER(x)                                      /* do nothing */
#else

/*
 * This is the semi-ANSI standard way of indicating that an
 * unused function parameter is required.
 */
#define UNUSED_PARAMETER(x)            (void) (x)
#endif
#endif
#endif                                 /* RTW_HEADER_rt_defines_h_ */
```

#### rtwtypes.h
```c
/*
 * rtwtypes.h
 *
 * Academic License - for use in teaching, academic research, and meeting
 * course requirements at degree granting institutions only.  Not for
 * government, commercial, or other organizational use.
 *
 * Code generation for model "reg_FF_PI_pl_regr_stiff".
 *
 * Model version              : 1.154
 * Simulink Coder version : 9.6 (R2021b) 14-May-2021
 * C source code generated on : Mon Jun 26 09:10:26 2023
 *
 * Target selection: bur_grt.tlc
 * Note: GRT includes extra infrastructure and instrumentation for prototyping
 * Embedded hardware selection: Intel->x86/Pentium
 * Code generation objectives: Unspecified
 * Validation result: Not run
 */

#ifndef RTWTYPES_H
#define RTWTYPES_H
#include "tmwtypes.h"
#ifndef POINTER_T
#define POINTER_T

typedef void * pointer_T;

#endif

/* Logical type definitions */
#if (!defined(__cplusplus))
#ifndef false
#define false                          (0U)
#endif

#ifndef true
#define true                           (1U)
#endif
#endif
#endif                                 /* RTWTYPES_H */
```

#### FF_PID_r.c
```c
/********************************************************************
 * COPYRIGHT -- B&R Industrial Automation GmbH
 ********************************************************************
 * Program: regulatory
 * File: regulatory.c
 * Author: MartinV
 * Last modified by: MartinV
 * Created: 12-Apr-2022 13:40:36
 * Last modified: Tue Apr 12 13:40:07 2022
 * Model Version: 1.105
 * Description:
 * modified Comment:
 ********************************************************************
 * Implementation of program regulatory
 ********************************************************************
 * Generated with B&R Automation Studio Target for Simulink V6.5
 * (GRT based)
 ********************************************************************/

#include <bur/plctypes.h>

#include "rtwtypes.h"
#include "rtmodel.h"

#define EXPAND_CONCAT(name1,name2) name1 ## name2
#define CONCAT(name1,name2) EXPAND_CONCAT(name1,name2)
#define RT_MODEL            CONCAT(MODEL,_rtModel)

#ifdef __cplusplus

extern "C" {

#endif

/* Defines */
#define SS_TERMINATE 4
#define SS_OUTPUT 3
#define SS_INITIALIZE 2

#ifdef __cplusplus

}

#endif

#ifdef __cplusplus
    unsigned long bur_heap_size = 6553500;
#endif

void FF_PID_r(struct FF_PID_r* inst)
{
  tag_RTM_regulator_FF_PI_plane_T* const regulator_FF_PI_plane_regres_M = &(inst)->bur_regulator_FF_PI_plane_regre;
	inst->bur_regulator_FF_PI_plane_regre.blockIO = &(inst)->bur_B_regulator_FF_PI_plane_reg;
	inst->bur_regulator_FF_PI_plane_regre.dwork = &(inst)->bur_DW_regulator_FF_PI_plane_re;

  switch (inst->ssMethodType)
  {
    case SS_INITIALIZE:

      /* call model initialize functions */
		/*memInit function */
		regulator_FF_PI_plane_regress_initializeMemory(regulator_FF_PI_plane_regres_M, inst);
		regulator_FF_PI_plane_regress_initialize(regulator_FF_PI_plane_regres_M, inst);
      break;

    case SS_OUTPUT:
      /* call model step functions */
		regulator_FF_PI_plane_regress_step(regulator_FF_PI_plane_regres_M, inst);
      break;

    case SS_TERMINATE:
      /* call model terminate function */
		regulator_FF_PI_plane_regress_terminate(regulator_FF_PI_plane_regres_M, inst);
	  break;
  }
}

/*****************************************************************************
   Function block sample time: 0.002
 *****************************************************************************/

/*****************************************************************************
   B&R Automation Studio Target for Simulink Version: V6.5.1 (03-Dec-2021)
 *****************************************************************************/
```

#### FF_PID_r_t.c
```c
/********************************************************************
 * COPYRIGHT -- B&R Industrial Automation GmbH
 ********************************************************************
 * Program: regulatory
 * File: regulatory.c
 * Author: MartinV
 * Last modified by: MartinV
 * Created: 26-Jun-2023 09:10:34
 * Last modified: Wed Jun 21 13:14:00 2023
 * Model Version: 1.154
 * Description:
 * modified Comment:
 ********************************************************************
 * Implementation of program regulatory
 ********************************************************************
 * Generated with B&R Automation Studio Target for Simulink V6.5
 * (GRT based)
 ********************************************************************/

#include <bur/plctypes.h>

#include "rtwtypes.h"
#include "rtmodel.h"

#define EXPAND_CONCAT(name1,name2) name1 ## name2
#define CONCAT(name1,name2) EXPAND_CONCAT(name1,name2)
#define RT_MODEL            CONCAT(MODEL,_rtModel)

#ifdef __cplusplus

extern "C" {

#endif

/* Defines */
#define SS_TERMINATE 4
#define SS_OUTPUT 3
#define SS_INITIALIZE 2

#ifdef __cplusplus

}

#endif

#ifdef __cplusplus
    unsigned long bur_heap_size = 6553500;
#endif

void FF_PID_r_t(struct FF_PID_r_t* inst)
{
  tag_RTM_reg_FF_PI_pl_regr_sti_T* const reg_FF_PI_pl_regr_stiff_M = &(inst)->bur_reg_FF_PI_pl_regr_stiff;
	inst->bur_reg_FF_PI_pl_regr_stiff.blockIO = &(inst)->bur_B_reg_FF_PI_pl_regr_stiff_T;
	inst->bur_reg_FF_PI_pl_regr_stiff.dwork = &(inst)->bur_DW_reg_FF_PI_pl_regr_stiff_;

  switch (inst->ssMethodType)
  {
    case SS_INITIALIZE:

      /* call model initialize functions */
		/*memInit function */
		reg_FF_PI_pl_regr_stiff_initializeMemory(reg_FF_PI_pl_regr_stiff_M, inst);
		reg_FF_PI_pl_regr_stiff_initialize(reg_FF_PI_pl_regr_stiff_M, inst);
      break;

    case SS_OUTPUT:
      /* call model step functions */
		reg_FF_PI_pl_regr_stiff_step(reg_FF_PI_pl_regr_stiff_M, inst);
      break;

    case SS_TERMINATE:
      /* call model terminate function */
		reg_FF_PI_pl_regr_stiff_terminate(reg_FF_PI_pl_regr_stiff_M, inst);
	  break;
  }
}

/*****************************************************************************
   Function block sample time: 0.002
 *****************************************************************************/

/*****************************************************************************
   B&R Automation Studio Target for Simulink Version: V6.5.1 (03-Dec-2021)
 *****************************************************************************/
```

#### reg_FF_PI_pl_regr_stiff.c
```c
/*
 * reg_FF_PI_pl_regr_stiff.c
 *
 * Academic License - for use in teaching, academic research, and meeting
 * course requirements at degree granting institutions only.  Not for
 * government, commercial, or other organizational use.
 *
 * Code generation for model "reg_FF_PI_pl_regr_stiff".
 *
 * Model version              : 1.154
 * Simulink Coder version : 9.6 (R2021b) 14-May-2021
 * C source code generated on : Mon Jun 26 09:10:26 2023
 *
 * Target selection: bur_grt.tlc
 * Note: GRT includes extra infrastructure and instrumentation for prototyping
 * Embedded hardware selection: Intel->x86/Pentium
 * Code generation objectives: Unspecified
 * Validation result: Not run
 */

#include "reg_FF_PI_pl_regr_stiff.h"
#include "reg_FF_PI_pl_regr_stiff_private.h"

/* Forward declaration for local functions */
static real32_T reg_FF_PI_pl_regr_stiff_norm(const real32_T x[4], struct FF_PID_r_t* inst);

/* Function for MATLAB Function: '<S4>/requested alfa 2 deltaz1' */
static real32_T reg_FF_PI_pl_regr_stiff_norm(const real32_T x[4], struct FF_PID_r_t* inst)
{
  real32_T absxk;
  real32_T scale;
  real32_T t;
  real32_T y;
  scale = 1.29246971E-26F;
  absxk = fabsf(x[0]);
  if (absxk > 1.29246971E-26F) {
    y = 1.0F;
    scale = absxk;
  } else {
    t = absxk / 1.29246971E-26F;
    y = t * t;
  }

  absxk = fabsf(x[1]);
  if (absxk > scale) {
    t = scale / absxk;
    y = y * t * t + 1.0F;
    scale = absxk;
  } else {
    t = absxk / scale;
    y += t * t;
  }

  absxk = fabsf(x[2]);
  if (absxk > scale) {
    t = scale / absxk;
    y = y * t * t + 1.0F;
    scale = absxk;
  } else {
    t = absxk / scale;
    y += t * t;
  }

  absxk = fabsf(x[3]);
  if (absxk > scale) {
    t = scale / absxk;
    y = y * t * t + 1.0F;
    scale = absxk;
  } else {
    t = absxk / scale;
    y += t * t;
  }

  return scale * sqrtf(y);
}

/* Model step function */
void reg_FF_PI_pl_regr_stiff_step(RT_MODEL_reg_FF_PI_pl_regr_st_T *const
  reg_FF_PI_pl_regr_stiff_M, struct FF_PID_r_t* inst)
{
  B_reg_FF_PI_pl_regr_stiff_T *reg_FF_PI_pl_regr_stiff_B =
    reg_FF_PI_pl_regr_stiff_M->blockIO;
  DW_reg_FF_PI_pl_regr_stiff_T *reg_FF_PI_pl_regr_stiff_DW =
    reg_FF_PI_pl_regr_stiff_M->dwork;
  real_T rtb_MultiportSwitch[48];
  real_T rtb_MultiportSwitch1[48];
  real_T rtb_MultiportSwitch2[48];
  real_T Blue0_tmp[4];
  real_T Yellow0_tmp[4];
  real_T A1;
  real_T A2;
  real_T A3;
  real_T rtb_Sum1;
  real_T rtb_Sum2;
  real_T rtb_Sum_d;
  real_T rtb_Switch1;
  int32_T Tz23_tmp;
  int32_T Tz23_tmp_tmp;
  int32_T i;
  int32_T i_0;
  real32_T AlphaY_0[16];
  real32_T HTransform[16];
  real32_T HTransform_tmp_2[16];
  real32_T Tz23_0[16];
  real32_T tmp[8];
  real32_T rtb_MultiportSwitch_0[6];
  real32_T tmp_0[6];
  real32_T Blue0_tmp_0[4];
  real32_T Green0_tmp_tmp_0[4];
  real32_T Yellow0_tmp_0[4];
  real32_T AlphaX;
  real32_T AlphaY;
  real32_T HTransform_tmp;
  real32_T rtb_Blue_real;
  real32_T rtb_Blue_ref;
  real32_T rtb_Green_ref;
  real32_T rtb_MultiportSwitch2_0;
  real32_T rtb_MultiportSwitch_1;
  real32_T rtb_MultiportSwitch_2;
  real32_T rtb_MultiportSwitch_3;
  real32_T rtb_MultiportSwitch_4;
  real32_T rtb_MultiportSwitch_5;
  real32_T rtb_MultiportSwitch_6;
  real32_T rtb_Yellow_real;
  real32_T rtb_Yellow_ref;
  real32_T tmp_1;
  real32_T tmp_2;
  int8_T Tz23[16];
  int8_T Green0_tmp_tmp[4];
  int8_T HTransform_tmp_0[4];
  int8_T HTransform_tmp_1[4];

  /* S-Function (bur_in): '<Root>/Input15' */
  reg_FF_PI_pl_regr_stiff_B->Input15 = inst->stiffness_ff;

  /* S-Function (bur_in): '<Root>/Input1' */
  reg_FF_PI_pl_regr_stiff_B->Input1 = inst->ref_alfa_x;

  /* S-Function (bur_in): '<Root>/Input2' */
  reg_FF_PI_pl_regr_stiff_B->Input2 = inst->ref_alfa_y;

  /* S-Function (bur_in): '<Root>/Input3' */
  reg_FF_PI_pl_regr_stiff_B->Input3 = inst->real_alfa_x;

  /* S-Function (bur_in): '<Root>/Input4' */
  reg_FF_PI_pl_regr_stiff_B->Input4 = inst->real_alfa_y;

  /* S-Function (bur_in): '<Root>/Input16' */
  reg_FF_PI_pl_regr_stiff_B->Input16 = inst->poradie_vlnovcov;

  /* MATLAB Function: '<S4>/requested alfa 2 deltaz1' incorporates:
   *  Constant: '<S4>/Constant1'
   */
  AlphaX = reg_FF_PI_pl_regr_stiff_B->Input1 * 3.14159274F / 180.0F;
  AlphaY = -reg_FF_PI_pl_regr_stiff_B->Input2 * 3.14159274F / 180.0F;
  Tz23[2] = 0;
  Tz23[6] = 0;
  Tz23[10] = 1;
  Tz23[14] = 80;
  HTransform_tmp = sinf(AlphaY);
  AlphaY = cosf(AlphaY);
  rtb_Blue_real = sinf(AlphaX);
  AlphaX = cosf(AlphaX);
  AlphaY_0[0] = AlphaY;
  AlphaY_0[4] = 0.0F;
  AlphaY_0[8] = HTransform_tmp;
  AlphaY_0[12] = 0.0F;
  AlphaY_0[2] = -HTransform_tmp;
  AlphaY_0[6] = 0.0F;
  AlphaY_0[10] = AlphaY;
  AlphaY_0[14] = 0.0F;
  Tz23[0] = 1;
  Tz23[1] = 0;
  Tz23[3] = 0;
  HTransform_tmp_1[0] = 1;
  AlphaY_0[1] = 0.0F;
  AlphaY_0[3] = 0.0F;
  HTransform_tmp_0[0] = 0;
  Tz23[4] = 0;
  Tz23[5] = 1;
  Tz23[7] = 0;
  HTransform_tmp_1[1] = 0;
  AlphaY_0[5] = 1.0F;
  AlphaY_0[7] = 0.0F;
  HTransform_tmp_0[1] = 0;
  Tz23[8] = 0;
  Tz23[9] = 0;
  Tz23[11] = 0;
  HTransform_tmp_1[2] = 0;
  AlphaY_0[9] = 0.0F;
  AlphaY_0[11] = 0.0F;
  HTransform_tmp_0[2] = 0;
  Tz23[12] = 0;
  Tz23[13] = 0;
  Tz23[15] = 1;
  HTransform_tmp_1[3] = 0;
  AlphaY_0[13] = 0.0F;
  AlphaY_0[15] = 1.0F;
  HTransform_tmp_0[3] = 1;
  HTransform_tmp_2[1] = 0.0F;
  HTransform_tmp_2[5] = AlphaX;
  HTransform_tmp_2[9] = -rtb_Blue_real;
  HTransform_tmp_2[13] = 0.0F;
  HTransform_tmp_2[2] = 0.0F;
  HTransform_tmp_2[6] = rtb_Blue_real;
  HTransform_tmp_2[10] = AlphaX;
  HTransform_tmp_2[14] = 0.0F;
  for (i = 0; i < 4; i++) {
    for (i_0 = 0; i_0 < 4; i_0++) {
      Tz23_tmp_tmp = i_0 << 2;
      Tz23_tmp = i + Tz23_tmp_tmp;
      Tz23_0[Tz23_tmp] = 0.0F;
      Tz23_0[Tz23_tmp] += AlphaY_0[Tz23_tmp_tmp] * (real32_T)Tz23[i];
      Tz23_0[Tz23_tmp] += AlphaY_0[Tz23_tmp_tmp + 1] * (real32_T)Tz23[i + 4];
      Tz23_0[Tz23_tmp] += AlphaY_0[Tz23_tmp_tmp + 2] * (real32_T)Tz23[i + 8];
      Tz23_0[Tz23_tmp] += AlphaY_0[Tz23_tmp_tmp + 3] * (real32_T)Tz23[i + 12];
    }

    Tz23_tmp_tmp = i << 2;
    HTransform_tmp_2[Tz23_tmp_tmp] = HTransform_tmp_1[i];
    HTransform_tmp_2[Tz23_tmp_tmp + 3] = HTransform_tmp_0[i];
  }

  for (i = 0; i < 4; i++) {
    for (i_0 = 0; i_0 < 4; i_0++) {
      Tz23_tmp_tmp = i_0 << 2;
      Tz23_tmp = i + Tz23_tmp_tmp;
      AlphaY_0[Tz23_tmp] = 0.0F;
      AlphaY_0[Tz23_tmp] += HTransform_tmp_2[Tz23_tmp_tmp] * Tz23_0[i];
      AlphaY_0[Tz23_tmp] += HTransform_tmp_2[Tz23_tmp_tmp + 1] * Tz23_0[i + 4];
      AlphaY_0[Tz23_tmp] += HTransform_tmp_2[Tz23_tmp_tmp + 2] * Tz23_0[i + 8];
      AlphaY_0[Tz23_tmp] += HTransform_tmp_2[Tz23_tmp_tmp + 3] * Tz23_0[i + 12];
    }

    for (i_0 = 0; i_0 < 4; i_0++) {
      Tz23_tmp_tmp = i_0 << 2;
      Tz23_tmp = i + Tz23_tmp_tmp;
      HTransform[Tz23_tmp] = 0.0F;
      HTransform[Tz23_tmp] += (real32_T)Tz23[Tz23_tmp_tmp] * AlphaY_0[i];
      HTransform[Tz23_tmp] += (real32_T)Tz23[Tz23_tmp_tmp + 1] * AlphaY_0[i + 4];
      HTransform[Tz23_tmp] += (real32_T)Tz23[Tz23_tmp_tmp + 2] * AlphaY_0[i + 8];
      HTransform[Tz23_tmp] += (real32_T)Tz23[Tz23_tmp_tmp + 3] * AlphaY_0[i + 12];
    }
  }

  Green0_tmp_tmp[0] = 107;
  Green0_tmp_tmp[1] = 0;
  Green0_tmp_tmp[2] = 0;
  Green0_tmp_tmp[3] = 1;
  Yellow0_tmp[0] = -53.5;
  Yellow0_tmp[1] = 92.664718204934928;
  Yellow0_tmp[2] = 0.0;
  Yellow0_tmp[3] = 1.0;
  Blue0_tmp[0] = -53.5;
  Blue0_tmp[1] = -92.664718204934928;
  Blue0_tmp[2] = 0.0;
  Blue0_tmp[3] = 1.0;
  switch ((int32_T)reg_FF_PI_pl_regr_stiff_B->Input16) {
   case 1:
    for (i = 0; i < 4; i++) {
      HTransform_tmp = HTransform[i + 12];
      Green0_tmp_tmp_0[i] = (real32_T)Green0_tmp_tmp[i] - (HTransform[i] *
        107.0F + HTransform_tmp);
      AlphaY = HTransform[i + 4];
      Blue0_tmp_0[i] = (real32_T)Blue0_tmp[i] - ((AlphaY * -92.6647186F +
        HTransform[i] * -53.5F) + HTransform_tmp);
      Yellow0_tmp_0[i] = (real32_T)Yellow0_tmp[i] - ((AlphaY * 92.6647186F +
        HTransform[i] * -53.5F) + HTransform_tmp);
    }

    rtb_Green_ref = reg_FF_PI_pl_regr_stiff_norm(Green0_tmp_tmp_0, inst);
    rtb_Blue_ref = reg_FF_PI_pl_regr_stiff_norm(Blue0_tmp_0, inst);
    rtb_Yellow_ref = reg_FF_PI_pl_regr_stiff_norm(Yellow0_tmp_0, inst);
    break;

   case 2:
    for (i = 0; i < 4; i++) {
      HTransform_tmp = HTransform[i + 12];
      Green0_tmp_tmp_0[i] = (real32_T)Green0_tmp_tmp[i] - (HTransform[i] *
        107.0F + HTransform_tmp);
      AlphaY = HTransform[i + 4];
      Yellow0_tmp_0[i] = (real32_T)Yellow0_tmp[i] - ((AlphaY * 92.6647186F +
        HTransform[i] * -53.5F) + HTransform_tmp);
      Blue0_tmp_0[i] = (real32_T)Blue0_tmp[i] - ((AlphaY * -92.6647186F +
        HTransform[i] * -53.5F) + HTransform_tmp);
    }

    rtb_Green_ref = reg_FF_PI_pl_regr_stiff_norm(Green0_tmp_tmp_0, inst);
    rtb_Blue_ref = reg_FF_PI_pl_regr_stiff_norm(Yellow0_tmp_0, inst);
    rtb_Yellow_ref = reg_FF_PI_pl_regr_stiff_norm(Blue0_tmp_0, inst);
    break;

   case 3:
    for (i = 0; i < 4; i++) {
      AlphaY = HTransform[i + 4];
      HTransform_tmp = HTransform[i + 12];
      Blue0_tmp_0[i] = (real32_T)Blue0_tmp[i] - ((AlphaY * -92.6647186F +
        HTransform[i] * -53.5F) + HTransform_tmp);
      Yellow0_tmp_0[i] = (real32_T)Yellow0_tmp[i] - ((AlphaY * 92.6647186F +
        HTransform[i] * -53.5F) + HTransform_tmp);
      Green0_tmp_tmp_0[i] = (real32_T)Green0_tmp_tmp[i] - (HTransform[i] *
        107.0F + HTransform_tmp);
    }

    rtb_Green_ref = reg_FF_PI_pl_regr_stiff_norm(Blue0_tmp_0, inst);
    rtb_Blue_ref = reg_FF_PI_pl_regr_stiff_norm(Yellow0_tmp_0, inst);
    rtb_Yellow_ref = reg_FF_PI_pl_regr_stiff_norm(Green0_tmp_tmp_0, inst);
    break;

   case 4:
    for (i = 0; i < 4; i++) {
      AlphaY = HTransform[i + 12];
      HTransform_tmp = HTransform[i + 4];
      Blue0_tmp_0[i] = (real32_T)Blue0_tmp[i] - ((HTransform_tmp * -92.6647186F
        + HTransform[i] * -53.5F) + AlphaY);
      Green0_tmp_tmp_0[i] = (real32_T)Green0_tmp_tmp[i] - (HTransform[i] *
        107.0F + AlphaY);
      Yellow0_tmp_0[i] = (real32_T)Yellow0_tmp[i] - ((HTransform_tmp *
        92.6647186F + HTransform[i] * -53.5F) + AlphaY);
    }

    rtb_Green_ref = reg_FF_PI_pl_regr_stiff_norm(Blue0_tmp_0, inst);
    rtb_Blue_ref = reg_FF_PI_pl_regr_stiff_norm(Green0_tmp_tmp_0, inst);
    rtb_Yellow_ref = reg_FF_PI_pl_regr_stiff_norm(Yellow0_tmp_0, inst);
    break;

   case 5:
    for (i = 0; i < 4; i++) {
      AlphaY = HTransform[i + 12];
      HTransform_tmp = HTransform[i + 4];
      Yellow0_tmp_0[i] = (real32_T)Yellow0_tmp[i] - ((HTransform_tmp *
        92.6647186F + HTransform[i] * -53.5F) + AlphaY);
      Green0_tmp_tmp_0[i] = (real32_T)Green0_tmp_tmp[i] - (HTransform[i] *
        107.0F + AlphaY);
      Blue0_tmp_0[i] = (real32_T)Blue0_tmp[i] - ((HTransform_tmp * -92.6647186F
        + HTransform[i] * -53.5F) + AlphaY);
    }

    rtb_Green_ref = reg_FF_PI_pl_regr_stiff_norm(Yellow0_tmp_0, inst);
    rtb_Blue_ref = reg_FF_PI_pl_regr_stiff_norm(Green0_tmp_tmp_0, inst);
    rtb_Yellow_ref = reg_FF_PI_pl_regr_stiff_norm(Blue0_tmp_0, inst);
    break;

   default:
    for (i = 0; i < 4; i++) {
      AlphaY = HTransform[i + 4];
      HTransform_tmp = HTransform[i + 12];
      Yellow0_tmp_0[i] = (real32_T)Yellow0_tmp[i] - ((AlphaY * 92.6647186F +
        HTransform[i] * -53.5F) + HTransform_tmp);
      Blue0_tmp_0[i] = (real32_T)Blue0_tmp[i] - ((AlphaY * -92.6647186F +
        HTransform[i] * -53.5F) + HTransform_tmp);
      Green0_tmp_tmp_0[i] = (real32_T)Green0_tmp_tmp[i] - (HTransform[i] *
        107.0F + HTransform_tmp);
    }

    rtb_Green_ref = reg_FF_PI_pl_regr_stiff_norm(Yellow0_tmp_0, inst);
    rtb_Blue_ref = reg_FF_PI_pl_regr_stiff_norm(Blue0_tmp_0, inst);
    rtb_Yellow_ref = reg_FF_PI_pl_regr_stiff_norm(Green0_tmp_tmp_0, inst);
    break;
  }

  AlphaX = reg_FF_PI_pl_regr_stiff_B->Input3 * 3.14159274F / 180.0F;
  AlphaY = -reg_FF_PI_pl_regr_stiff_B->Input4 * 3.14159274F / 180.0F;
  HTransform_tmp = sinf(AlphaY);
  AlphaY = cosf(AlphaY);
  rtb_Blue_real = sinf(AlphaX);
  AlphaX = cosf(AlphaX);
  AlphaY_0[0] = AlphaY;
  AlphaY_0[4] = 0.0F;
  AlphaY_0[8] = HTransform_tmp;
  AlphaY_0[12] = 0.0F;
  AlphaY_0[2] = -HTransform_tmp;
  AlphaY_0[6] = 0.0F;
  AlphaY_0[10] = AlphaY;
  AlphaY_0[14] = 0.0F;
  AlphaY_0[1] = 0.0F;
  AlphaY_0[3] = 0.0F;
  AlphaY_0[5] = 1.0F;
  AlphaY_0[7] = 0.0F;
  AlphaY_0[9] = 0.0F;
  AlphaY_0[11] = 0.0F;
  AlphaY_0[13] = 0.0F;
  AlphaY_0[15] = 1.0F;
  HTransform_tmp_2[1] = 0.0F;
  HTransform_tmp_2[5] = AlphaX;
  HTransform_tmp_2[9] = -rtb_Blue_real;
  HTransform_tmp_2[13] = 0.0F;
  HTransform_tmp_2[2] = 0.0F;
  HTransform_tmp_2[6] = rtb_Blue_real;
  HTransform_tmp_2[10] = AlphaX;
  HTransform_tmp_2[14] = 0.0F;
  for (i = 0; i < 4; i++) {
    for (i_0 = 0; i_0 < 4; i_0++) {
      Tz23_tmp_tmp = i_0 << 2;
      Tz23_tmp = i + Tz23_tmp_tmp;
      Tz23_0[Tz23_tmp] = 0.0F;
      Tz23_0[Tz23_tmp] += AlphaY_0[Tz23_tmp_tmp] * (real32_T)Tz23[i];
      Tz23_0[Tz23_tmp] += AlphaY_0[Tz23_tmp_tmp + 1] * (real32_T)Tz23[i + 4];
      Tz23_0[Tz23_tmp] += AlphaY_0[Tz23_tmp_tmp + 2] * (real32_T)Tz23[i + 8];
      Tz23_0[Tz23_tmp] += AlphaY_0[Tz23_tmp_tmp + 3] * (real32_T)Tz23[i + 12];
    }

    Tz23_tmp_tmp = i << 2;
    HTransform_tmp_2[Tz23_tmp_tmp] = HTransform_tmp_1[i];
    HTransform_tmp_2[Tz23_tmp_tmp + 3] = HTransform_tmp_0[i];
  }

  Yellow0_tmp[0] = -53.5;
  Yellow0_tmp[1] = 92.664718204934928;
  Yellow0_tmp[2] = 0.0;
  Yellow0_tmp[3] = 1.0;
  Blue0_tmp[0] = -53.5;
  Blue0_tmp[1] = -92.664718204934928;
  Blue0_tmp[2] = 0.0;
  Blue0_tmp[3] = 1.0;
  for (i = 0; i < 4; i++) {
    for (i_0 = 0; i_0 < 4; i_0++) {
      Tz23_tmp_tmp = i_0 << 2;
      Tz23_tmp = i + Tz23_tmp_tmp;
      AlphaY_0[Tz23_tmp] = 0.0F;
      AlphaY_0[Tz23_tmp] += HTransform_tmp_2[Tz23_tmp_tmp] * Tz23_0[i];
      AlphaY_0[Tz23_tmp] += HTransform_tmp_2[Tz23_tmp_tmp + 1] * Tz23_0[i + 4];
      AlphaY_0[Tz23_tmp] += HTransform_tmp_2[Tz23_tmp_tmp + 2] * Tz23_0[i + 8];
      AlphaY_0[Tz23_tmp] += HTransform_tmp_2[Tz23_tmp_tmp + 3] * Tz23_0[i + 12];
    }

    AlphaY = 0.0F;
    HTransform_tmp = 0.0F;
    rtb_Blue_real = 0.0F;
    for (i_0 = 0; i_0 < 4; i_0++) {
      Tz23_tmp_tmp = i_0 << 2;
      Tz23_tmp = i + Tz23_tmp_tmp;
      HTransform[Tz23_tmp] = 0.0F;
      HTransform[Tz23_tmp] += (real32_T)Tz23[Tz23_tmp_tmp] * AlphaY_0[i];
      HTransform[Tz23_tmp] += (real32_T)Tz23[Tz23_tmp_tmp + 1] * AlphaY_0[i + 4];
      HTransform[Tz23_tmp] += (real32_T)Tz23[Tz23_tmp_tmp + 2] * AlphaY_0[i + 8];
      HTransform[Tz23_tmp] += (real32_T)Tz23[Tz23_tmp_tmp + 3] * AlphaY_0[i + 12];
      AlphaY += HTransform[Tz23_tmp] * (real32_T)Green0_tmp_tmp[i_0];
      HTransform_tmp += HTransform[Tz23_tmp] * (real32_T)Blue0_tmp[i_0];
      rtb_Blue_real += HTransform[Tz23_tmp] * (real32_T)Yellow0_tmp[i_0];
    }

    Green0_tmp_tmp_0[i] = (real32_T)Green0_tmp_tmp[i] - AlphaY;
    Blue0_tmp_0[i] = (real32_T)Blue0_tmp[i] - HTransform_tmp;
    Yellow0_tmp_0[i] = (real32_T)Yellow0_tmp[i] - rtb_Blue_real;
  }

  HTransform_tmp = reg_FF_PI_pl_regr_stiff_norm(Green0_tmp_tmp_0, inst);
  AlphaX = HTransform_tmp;
  AlphaY = reg_FF_PI_pl_regr_stiff_norm(Blue0_tmp_0, inst);
  rtb_Blue_real = AlphaY;
  rtb_Yellow_real = reg_FF_PI_pl_regr_stiff_norm(Yellow0_tmp_0, inst);
  switch ((int32_T)reg_FF_PI_pl_regr_stiff_B->Input16) {
   case 1:
    break;

   case 2:
    rtb_Blue_real = rtb_Yellow_real;
    rtb_Yellow_real = AlphaY;
    break;

   case 3:
    AlphaX = AlphaY;
    rtb_Blue_real = rtb_Yellow_real;
    rtb_Yellow_real = HTransform_tmp;
    break;

   case 4:
    rtb_Green_ref = AlphaY;
    rtb_Blue_ref = HTransform_tmp;
    rtb_Yellow_ref = rtb_Yellow_real;
    break;

   case 5:
    AlphaX = rtb_Yellow_real;
    rtb_Blue_real = HTransform_tmp;
    rtb_Yellow_real = AlphaY;
    break;

   default:
    AlphaX = rtb_Yellow_real;
    rtb_Yellow_real = HTransform_tmp;
    break;
  }

  /* End of MATLAB Function: '<S4>/requested alfa 2 deltaz1' */

  /* Sum: '<S2>/Sum' incorporates:
   *  Constant: '<S10>/cylinder height'
   *  Constant: '<S8>/cylinder height'
   *  Gain: '<S4>/Gain'
   *  Gain: '<S4>/Gain3'
   *  Sum: '<S10>/Sum'
   *  Sum: '<S8>/Sum'
   */
  A2 = (0.001F * rtb_Blue_real - 0.16) - (0.001F * rtb_Blue_ref - 0.16);

  /* S-Function (bur_in): '<Root>/Input11' */
  reg_FF_PI_pl_regr_stiff_B->Input11 = inst->P_parameter;

  /* S-Function (bur_in): '<Root>/Input5' */
  reg_FF_PI_pl_regr_stiff_B->Input5 = inst->reset_PID_blue;

  /* DiscreteIntegrator: '<S144>/Integrator' */
  if ((reg_FF_PI_pl_regr_stiff_B->Input5 <= 0.0F) &&
      (reg_FF_PI_pl_regr_stiff_DW->Integrator_PrevResetState == 1)) {
    reg_FF_PI_pl_regr_stiff_DW->Integrator_DSTATE = 0.0;
  }

  /* S-Function (bur_in): '<Root>/Input13' */
  reg_FF_PI_pl_regr_stiff_B->Input13 = inst->D_parameter;

  /* DiscreteIntegrator: '<S139>/Filter' */
  if ((reg_FF_PI_pl_regr_stiff_B->Input5 <= 0.0F) &&
      (reg_FF_PI_pl_regr_stiff_DW->Filter_PrevResetState == 1)) {
    reg_FF_PI_pl_regr_stiff_DW->Filter_DSTATE = 0.0;
  }

  /* S-Function (bur_in): '<Root>/Input14' */
  reg_FF_PI_pl_regr_stiff_B->Input14 = inst->N_parameter;

  /* Product: '<S147>/NProd Out' incorporates:
   *  DiscreteIntegrator: '<S139>/Filter'
   *  Product: '<S138>/DProd Out'
   *  Sum: '<S139>/SumD'
   */
  A1 = (A2 * reg_FF_PI_pl_regr_stiff_B->Input13 -
        reg_FF_PI_pl_regr_stiff_DW->Filter_DSTATE) *
    reg_FF_PI_pl_regr_stiff_B->Input14;

  /* Switch: '<Root>/Switch2' */
  if (reg_FF_PI_pl_regr_stiff_B->Input5 > 0.0F) {
    /* Sum: '<S154>/Sum' incorporates:
     *  DiscreteIntegrator: '<S144>/Integrator'
     *  Product: '<S149>/PProd Out'
     */
    A3 = (A2 * reg_FF_PI_pl_regr_stiff_B->Input11 +
          reg_FF_PI_pl_regr_stiff_DW->Integrator_DSTATE) + A1;

    /* Switch: '<S152>/Switch2' incorporates:
     *  Constant: '<S2>/max_sat'
     *  Constant: '<S2>/min_sat'
     *  RelationalOperator: '<S152>/LowerRelop1'
     *  RelationalOperator: '<S152>/UpperRelop'
     *  Sum: '<S2>/Sum3'
     *  Sum: '<S2>/Sum4'
     *  Switch: '<S152>/Switch'
     */
    if (A3 > 5.0 - reg_FF_PI_pl_regr_stiff_B->Input15) {
      rtb_Switch1 = 5.0 - reg_FF_PI_pl_regr_stiff_B->Input15;
    } else if (A3 < 0.0 - reg_FF_PI_pl_regr_stiff_B->Input15) {
      /* Switch: '<S152>/Switch' incorporates:
       *  Constant: '<S2>/min_sat'
       *  Sum: '<S2>/Sum4'
       */
      rtb_Switch1 = 0.0 - reg_FF_PI_pl_regr_stiff_B->Input15;
    } else {
      rtb_Switch1 = A3;
    }

    /* End of Switch: '<S152>/Switch2' */
  } else {
    rtb_Switch1 = 0.0;
  }

  /* End of Switch: '<Root>/Switch2' */

  /* S-Function (bur_in): '<Root>/Input17' */
  reg_FF_PI_pl_regr_stiff_B->Input17 = inst->platform_ID;

  /* MultiPortSwitch: '<S1>/Multiport Switch' incorporates:
   *  Constant: '<S1>/Constant'
   *  Constant: '<S1>/Constant2'
   *  Constant: '<S1>/Constant4'
   *  Constant: '<S1>/Constant5'
   *  Constant: '<S1>/Constant6'
   *  Constant: '<S1>/Constant7'
   */
  switch ((int32_T)reg_FF_PI_pl_regr_stiff_B->Input17) {
   case 1:
    for (i = 0; i < 48; i++) {
      rtb_MultiportSwitch[i] = reg_FF_PI_pl_regr_stiff_ConstP.Constant_Value[i];
    }
    break;

   case 2:
    for (i = 0; i < 48; i++) {
      rtb_MultiportSwitch[i] = reg_FF_PI_pl_regr_stiff_ConstP.Constant2_Value[i];
    }
    break;

   case 3:
    for (i = 0; i < 48; i++) {
      rtb_MultiportSwitch[i] = reg_FF_PI_pl_regr_stiff_ConstP.Constant4_Value[i];
    }
    break;

   case 4:
    for (i = 0; i < 48; i++) {
      rtb_MultiportSwitch[i] = reg_FF_PI_pl_regr_stiff_ConstP.pooled3[i];
    }
    break;

   case 5:
    for (i = 0; i < 48; i++) {
      rtb_MultiportSwitch[i] = reg_FF_PI_pl_regr_stiff_ConstP.pooled3[i];
    }
    break;

   default:
    for (i = 0; i < 48; i++) {
      rtb_MultiportSwitch[i] = reg_FF_PI_pl_regr_stiff_ConstP.pooled3[i];
    }
    break;
  }

  /* End of MultiPortSwitch: '<S1>/Multiport Switch' */

  /* MultiPortSwitch: '<S1>/Multiport Switch1' incorporates:
   *  Constant: '<S1>/Constant1'
   *  Constant: '<S1>/Constant10'
   *  Constant: '<S1>/Constant11'
   *  Constant: '<S1>/Constant12'
   *  Constant: '<S1>/Constant8'
   *  Constant: '<S1>/Constant9'
   */
  switch ((int32_T)reg_FF_PI_pl_regr_stiff_B->Input17) {
   case 1:
    for (i = 0; i < 48; i++) {
      rtb_MultiportSwitch1[i] = reg_FF_PI_pl_regr_stiff_ConstP.Constant1_Value[i];
    }
    break;

   case 2:
    for (i = 0; i < 48; i++) {
      rtb_MultiportSwitch1[i] = reg_FF_PI_pl_regr_stiff_ConstP.Constant8_Value[i];
    }
    break;

   case 3:
    for (i = 0; i < 48; i++) {
      rtb_MultiportSwitch1[i] = reg_FF_PI_pl_regr_stiff_ConstP.Constant9_Value[i];
    }
    break;

   case 4:
    for (i = 0; i < 48; i++) {
      rtb_MultiportSwitch1[i] = reg_FF_PI_pl_regr_stiff_ConstP.pooled1[i];
    }
    break;

   case 5:
    for (i = 0; i < 48; i++) {
      rtb_MultiportSwitch1[i] = reg_FF_PI_pl_regr_stiff_ConstP.pooled1[i];
    }
    break;

   default:
    for (i = 0; i < 48; i++) {
      rtb_MultiportSwitch1[i] = reg_FF_PI_pl_regr_stiff_ConstP.pooled1[i];
    }
    break;
  }

  /* End of MultiPortSwitch: '<S1>/Multiport Switch1' */

  /* MultiPortSwitch: '<S1>/Multiport Switch2' incorporates:
   *  Constant: '<S1>/Constant13'
   *  Constant: '<S1>/Constant14'
   *  Constant: '<S1>/Constant15'
   *  Constant: '<S1>/Constant16'
   *  Constant: '<S1>/Constant17'
   *  Constant: '<S1>/Constant3'
   */
  switch ((int32_T)reg_FF_PI_pl_regr_stiff_B->Input17) {
   case 1:
    for (i = 0; i < 48; i++) {
      rtb_MultiportSwitch2[i] = reg_FF_PI_pl_regr_stiff_ConstP.Constant3_Value[i];
    }
    break;

   case 2:
    for (i = 0; i < 48; i++) {
      rtb_MultiportSwitch2[i] =
        reg_FF_PI_pl_regr_stiff_ConstP.Constant13_Value[i];
    }
    break;

   case 3:
    for (i = 0; i < 48; i++) {
      rtb_MultiportSwitch2[i] =
        reg_FF_PI_pl_regr_stiff_ConstP.Constant14_Value[i];
    }
    break;

   case 4:
    for (i = 0; i < 48; i++) {
      rtb_MultiportSwitch2[i] = reg_FF_PI_pl_regr_stiff_ConstP.pooled2[i];
    }
    break;

   case 5:
    for (i = 0; i < 48; i++) {
      rtb_MultiportSwitch2[i] = reg_FF_PI_pl_regr_stiff_ConstP.pooled2[i];
    }
    break;

   default:
    for (i = 0; i < 48; i++) {
      rtb_MultiportSwitch2[i] = reg_FF_PI_pl_regr_stiff_ConstP.pooled2[i];
    }
    break;
  }

  /* End of MultiPortSwitch: '<S1>/Multiport Switch2' */

  /* MATLAB Function: '<S1>/MATLAB Function' incorporates:
   *  MultiPortSwitch: '<S1>/Multiport Switch'
   */
  AlphaY = powf(reg_FF_PI_pl_regr_stiff_B->Input15, 7.0F);
  tmp[0] = AlphaY;
  HTransform_tmp = powf(reg_FF_PI_pl_regr_stiff_B->Input15, 6.0F);
  tmp[1] = HTransform_tmp;
  rtb_Blue_real = powf(reg_FF_PI_pl_regr_stiff_B->Input15, 5.0F);
  tmp[2] = rtb_Blue_real;
  rtb_Blue_ref = powf(reg_FF_PI_pl_regr_stiff_B->Input15, 4.0F);
  tmp[3] = rtb_Blue_ref;
  tmp_1 = powf(reg_FF_PI_pl_regr_stiff_B->Input15, 3.0F);
  tmp[4] = tmp_1;
  tmp_2 = reg_FF_PI_pl_regr_stiff_B->Input15 *
    reg_FF_PI_pl_regr_stiff_B->Input15;
  tmp[5] = tmp_2;
  tmp[6] = reg_FF_PI_pl_regr_stiff_B->Input15;
  tmp[7] = 1.0F;
  rtb_MultiportSwitch_1 = 0.0F;
  for (i = 0; i < 8; i++) {
    rtb_MultiportSwitch_1 += (real32_T)rtb_MultiportSwitch[6 * i] * tmp[i];
  }

  tmp[0] = AlphaY;
  tmp[1] = HTransform_tmp;
  tmp[2] = rtb_Blue_real;
  tmp[3] = rtb_Blue_ref;
  tmp[4] = tmp_1;
  tmp[5] = tmp_2;
  tmp[6] = reg_FF_PI_pl_regr_stiff_B->Input15;
  tmp[7] = 1.0F;
  rtb_MultiportSwitch_2 = 0.0F;
  for (i = 0; i < 8; i++) {
    rtb_MultiportSwitch_2 += (real32_T)rtb_MultiportSwitch[6 * i + 1] * tmp[i];
  }

  tmp[0] = AlphaY;
  tmp[1] = HTransform_tmp;
  tmp[2] = rtb_Blue_real;
  tmp[3] = rtb_Blue_ref;
  tmp[4] = tmp_1;
  tmp[5] = tmp_2;
  tmp[6] = reg_FF_PI_pl_regr_stiff_B->Input15;
  tmp[7] = 1.0F;
  rtb_MultiportSwitch_3 = 0.0F;
  for (i = 0; i < 8; i++) {
    rtb_MultiportSwitch_3 += (real32_T)rtb_MultiportSwitch[6 * i + 2] * tmp[i];
  }

  tmp[0] = AlphaY;
  tmp[1] = HTransform_tmp;
  tmp[2] = rtb_Blue_real;
  tmp[3] = rtb_Blue_ref;
  tmp[4] = tmp_1;
  tmp[5] = tmp_2;
  tmp[6] = reg_FF_PI_pl_regr_stiff_B->Input15;
  tmp[7] = 1.0F;
  rtb_MultiportSwitch_4 = 0.0F;
  for (i = 0; i < 8; i++) {
    rtb_MultiportSwitch_4 += (real32_T)rtb_MultiportSwitch[6 * i + 3] * tmp[i];
  }

  tmp[0] = AlphaY;
  tmp[1] = HTransform_tmp;
  tmp[2] = rtb_Blue_real;
  tmp[3] = rtb_Blue_ref;
  tmp[4] = tmp_1;
  tmp[5] = tmp_2;
  tmp[6] = reg_FF_PI_pl_regr_stiff_B->Input15;
  tmp[7] = 1.0F;
  rtb_MultiportSwitch_5 = 0.0F;
  for (i = 0; i < 8; i++) {
    rtb_MultiportSwitch_5 += (real32_T)rtb_MultiportSwitch[6 * i + 4] * tmp[i];
  }

  tmp[0] = AlphaY;
  tmp[1] = HTransform_tmp;
  tmp[2] = rtb_Blue_real;
  tmp[3] = rtb_Blue_ref;
  tmp[4] = tmp_1;
  tmp[5] = tmp_2;
  tmp[6] = reg_FF_PI_pl_regr_stiff_B->Input15;
  tmp[7] = 1.0F;
  rtb_MultiportSwitch_6 = 0.0F;
  for (i = 0; i < 8; i++) {
    rtb_MultiportSwitch_6 += (real32_T)rtb_MultiportSwitch[6 * i + 5] * tmp[i];
  }

  rtb_MultiportSwitch_0[0] = rtb_MultiportSwitch_1;
  rtb_MultiportSwitch_0[1] = rtb_MultiportSwitch_2;
  rtb_MultiportSwitch_0[2] = rtb_MultiportSwitch_3;
  rtb_MultiportSwitch_0[3] = rtb_MultiportSwitch_4;
  rtb_MultiportSwitch_0[4] = rtb_MultiportSwitch_5;
  rtb_MultiportSwitch_0[5] = rtb_MultiportSwitch_6;
  tmp_0[0] = 1.0F;
  tmp_0[1] = reg_FF_PI_pl_regr_stiff_B->Input1;
  tmp_0[2] = reg_FF_PI_pl_regr_stiff_B->Input2;
  rtb_MultiportSwitch_2 = reg_FF_PI_pl_regr_stiff_B->Input1 *
    reg_FF_PI_pl_regr_stiff_B->Input1;
  tmp_0[3] = rtb_MultiportSwitch_2;
  rtb_MultiportSwitch_3 = reg_FF_PI_pl_regr_stiff_B->Input1 *
    reg_FF_PI_pl_regr_stiff_B->Input2;
  tmp_0[4] = rtb_MultiportSwitch_3;
  rtb_MultiportSwitch_4 = reg_FF_PI_pl_regr_stiff_B->Input2 *
    reg_FF_PI_pl_regr_stiff_B->Input2;
  tmp_0[5] = rtb_MultiportSwitch_4;
  rtb_MultiportSwitch_1 = 0.0F;
  for (i = 0; i < 6; i++) {
    rtb_MultiportSwitch_1 += rtb_MultiportSwitch_0[i] * tmp_0[i];
  }

  /* Sum: '<Root>/Sum' incorporates:
   *  MATLAB Function: '<S1>/MATLAB Function'
   */
  reg_FF_PI_pl_regr_stiff_B->Sum = (real32_T)(rtb_Switch1 +
    rtb_MultiportSwitch_1);

  /* S-Function (bur_out): '<Root>/Output1' */
  inst->Blue_tab = reg_FF_PI_pl_regr_stiff_B->Sum;

  /* Sum: '<S2>/Sum2' incorporates:
   *  Constant: '<S11>/cylinder height'
   *  Constant: '<S13>/cylinder height'
   *  Gain: '<S4>/Gain1'
   *  Gain: '<S4>/Gain4'
   *  Sum: '<S11>/Sum'
   *  Sum: '<S13>/Sum'
   */
  rtb_Sum2 = (0.001F * AlphaX - 0.16) - (0.001F * rtb_Green_ref - 0.16);

  /* S-Function (bur_in): '<Root>/Input7' */
  reg_FF_PI_pl_regr_stiff_B->Input7 = inst->reset_PID_green;

  /* DiscreteIntegrator: '<S95>/Integrator' */
  if ((reg_FF_PI_pl_regr_stiff_B->Input7 <= 0.0F) &&
      (reg_FF_PI_pl_regr_stiff_DW->Integrator_PrevResetState_l == 1)) {
    reg_FF_PI_pl_regr_stiff_DW->Integrator_DSTATE_o = 0.0;
  }

  /* DiscreteIntegrator: '<S90>/Filter' */
  if ((reg_FF_PI_pl_regr_stiff_B->Input7 <= 0.0F) &&
      (reg_FF_PI_pl_regr_stiff_DW->Filter_PrevResetState_e == 1)) {
    reg_FF_PI_pl_regr_stiff_DW->Filter_DSTATE_f = 0.0;
  }

  /* Product: '<S98>/NProd Out' incorporates:
   *  DiscreteIntegrator: '<S90>/Filter'
   *  Product: '<S89>/DProd Out'
   *  Sum: '<S90>/SumD'
   */
  A3 = (rtb_Sum2 * reg_FF_PI_pl_regr_stiff_B->Input13 -
        reg_FF_PI_pl_regr_stiff_DW->Filter_DSTATE_f) *
    reg_FF_PI_pl_regr_stiff_B->Input14;

  /* Switch: '<Root>/Switch' */
  if (reg_FF_PI_pl_regr_stiff_B->Input7 > 0.0F) {
    /* Sum: '<S105>/Sum' incorporates:
     *  DiscreteIntegrator: '<S95>/Integrator'
     *  Product: '<S100>/PProd Out'
     */
    rtb_Sum_d = (rtb_Sum2 * reg_FF_PI_pl_regr_stiff_B->Input11 +
                 reg_FF_PI_pl_regr_stiff_DW->Integrator_DSTATE_o) + A3;

    /* Switch: '<S103>/Switch2' incorporates:
     *  Constant: '<S2>/max_sat'
     *  Constant: '<S2>/min_sat'
     *  RelationalOperator: '<S103>/LowerRelop1'
     *  RelationalOperator: '<S103>/UpperRelop'
     *  Sum: '<S2>/Sum3'
     *  Sum: '<S2>/Sum4'
     *  Switch: '<S103>/Switch'
     */
    if (rtb_Sum_d > 5.0 - reg_FF_PI_pl_regr_stiff_B->Input15) {
      rtb_Switch1 = 5.0 - reg_FF_PI_pl_regr_stiff_B->Input15;
    } else if (rtb_Sum_d < 0.0 - reg_FF_PI_pl_regr_stiff_B->Input15) {
      /* Switch: '<S103>/Switch' incorporates:
       *  Constant: '<S2>/min_sat'
       *  Sum: '<S2>/Sum4'
       */
      rtb_Switch1 = 0.0 - reg_FF_PI_pl_regr_stiff_B->Input15;
    } else {
      rtb_Switch1 = rtb_Sum_d;
    }

    /* End of Switch: '<S103>/Switch2' */
  } else {
    rtb_Switch1 = 0.0;
  }

  /* End of Switch: '<Root>/Switch' */

  /* MATLAB Function: '<S1>/MATLAB Function' incorporates:
   *  MultiPortSwitch: '<S1>/Multiport Switch2'
   */
  tmp[0] = AlphaY;
  tmp[1] = HTransform_tmp;
  tmp[2] = rtb_Blue_real;
  tmp[3] = rtb_Blue_ref;
  tmp[4] = tmp_1;
  tmp[5] = tmp_2;
  tmp[6] = reg_FF_PI_pl_regr_stiff_B->Input15;
  tmp[7] = 1.0F;
  AlphaX = 0.0F;
  for (i = 0; i < 8; i++) {
    AlphaX += (real32_T)rtb_MultiportSwitch2[6 * i] * tmp[i];
  }

  tmp[0] = AlphaY;
  tmp[1] = HTransform_tmp;
  tmp[2] = rtb_Blue_real;
  tmp[3] = rtb_Blue_ref;
  tmp[4] = tmp_1;
  tmp[5] = tmp_2;
  tmp[6] = reg_FF_PI_pl_regr_stiff_B->Input15;
  tmp[7] = 1.0F;
  rtb_Green_ref = 0.0F;
  for (i = 0; i < 8; i++) {
    rtb_Green_ref += (real32_T)rtb_MultiportSwitch2[6 * i + 1] * tmp[i];
  }

  tmp[0] = AlphaY;
  tmp[1] = HTransform_tmp;
  tmp[2] = rtb_Blue_real;
  tmp[3] = rtb_Blue_ref;
  tmp[4] = tmp_1;
  tmp[5] = tmp_2;
  tmp[6] = reg_FF_PI_pl_regr_stiff_B->Input15;
  tmp[7] = 1.0F;
  rtb_MultiportSwitch_1 = 0.0F;
  for (i = 0; i < 8; i++) {
    rtb_MultiportSwitch_1 += (real32_T)rtb_MultiportSwitch2[6 * i + 2] * tmp[i];
  }

  tmp[0] = AlphaY;
  tmp[1] = HTransform_tmp;
  tmp[2] = rtb_Blue_real;
  tmp[3] = rtb_Blue_ref;
  tmp[4] = tmp_1;
  tmp[5] = tmp_2;
  tmp[6] = reg_FF_PI_pl_regr_stiff_B->Input15;
  tmp[7] = 1.0F;
  rtb_MultiportSwitch_5 = 0.0F;
  for (i = 0; i < 8; i++) {
    rtb_MultiportSwitch_5 += (real32_T)rtb_MultiportSwitch2[6 * i + 3] * tmp[i];
  }

  tmp[0] = AlphaY;
  tmp[1] = HTransform_tmp;
  tmp[2] = rtb_Blue_real;
  tmp[3] = rtb_Blue_ref;
  tmp[4] = tmp_1;
  tmp[5] = tmp_2;
  tmp[6] = reg_FF_PI_pl_regr_stiff_B->Input15;
  tmp[7] = 1.0F;
  rtb_MultiportSwitch_6 = 0.0F;
  for (i = 0; i < 8; i++) {
    rtb_MultiportSwitch_6 += (real32_T)rtb_MultiportSwitch2[6 * i + 4] * tmp[i];
  }

  tmp[0] = AlphaY;
  tmp[1] = HTransform_tmp;
  tmp[2] = rtb_Blue_real;
  tmp[3] = rtb_Blue_ref;
  tmp[4] = tmp_1;
  tmp[5] = tmp_2;
  tmp[6] = reg_FF_PI_pl_regr_stiff_B->Input15;
  tmp[7] = 1.0F;
  rtb_MultiportSwitch2_0 = 0.0F;
  for (i = 0; i < 8; i++) {
    rtb_MultiportSwitch2_0 += (real32_T)rtb_MultiportSwitch2[6 * i + 5] * tmp[i];
  }

  rtb_MultiportSwitch_0[0] = AlphaX;
  rtb_MultiportSwitch_0[1] = rtb_Green_ref;
  rtb_MultiportSwitch_0[2] = rtb_MultiportSwitch_1;
  rtb_MultiportSwitch_0[3] = rtb_MultiportSwitch_5;
  rtb_MultiportSwitch_0[4] = rtb_MultiportSwitch_6;
  rtb_MultiportSwitch_0[5] = rtb_MultiportSwitch2_0;
  tmp_0[0] = 1.0F;
  tmp_0[1] = reg_FF_PI_pl_regr_stiff_B->Input1;
  tmp_0[2] = reg_FF_PI_pl_regr_stiff_B->Input2;
  tmp_0[3] = rtb_MultiportSwitch_2;
  tmp_0[4] = rtb_MultiportSwitch_3;
  tmp_0[5] = rtb_MultiportSwitch_4;
  AlphaX = 0.0F;
  for (i = 0; i < 6; i++) {
    AlphaX += rtb_MultiportSwitch_0[i] * tmp_0[i];
  }

  /* Sum: '<Root>/Sum2' incorporates:
   *  MATLAB Function: '<S1>/MATLAB Function'
   */
  reg_FF_PI_pl_regr_stiff_B->Sum2 = (real32_T)(rtb_Switch1 + AlphaX);

  /* S-Function (bur_out): '<Root>/Output2' */
  inst->Yellow_tab = reg_FF_PI_pl_regr_stiff_B->Sum2;

  /* Sum: '<S2>/Sum1' incorporates:
   *  Constant: '<S12>/cylinder height'
   *  Constant: '<S9>/cylinder height'
   *  Gain: '<S4>/Gain2'
   *  Gain: '<S4>/Gain5'
   *  Sum: '<S12>/Sum'
   *  Sum: '<S9>/Sum'
   */
  rtb_Sum1 = (0.001F * rtb_Yellow_real - 0.16) - (0.001F * rtb_Yellow_ref - 0.16);

  /* S-Function (bur_in): '<Root>/Input6' */
  reg_FF_PI_pl_regr_stiff_B->Input6 = inst->reset_PID_yellow;

  /* DiscreteIntegrator: '<S46>/Integrator' */
  if ((reg_FF_PI_pl_regr_stiff_B->Input6 <= 0.0F) &&
      (reg_FF_PI_pl_regr_stiff_DW->Integrator_PrevResetState_e == 1)) {
    reg_FF_PI_pl_regr_stiff_DW->Integrator_DSTATE_i = 0.0;
  }

  /* DiscreteIntegrator: '<S41>/Filter' */
  if ((reg_FF_PI_pl_regr_stiff_B->Input6 <= 0.0F) &&
      (reg_FF_PI_pl_regr_stiff_DW->Filter_PrevResetState_h == 1)) {
    reg_FF_PI_pl_regr_stiff_DW->Filter_DSTATE_a = 0.0;
  }

  /* Product: '<S49>/NProd Out' incorporates:
   *  DiscreteIntegrator: '<S41>/Filter'
   *  Product: '<S40>/DProd Out'
   *  Sum: '<S41>/SumD'
   */
  rtb_Sum_d = (rtb_Sum1 * reg_FF_PI_pl_regr_stiff_B->Input13 -
               reg_FF_PI_pl_regr_stiff_DW->Filter_DSTATE_a) *
    reg_FF_PI_pl_regr_stiff_B->Input14;

  /* Switch: '<Root>/Switch1' */
  if (reg_FF_PI_pl_regr_stiff_B->Input6 > 0.0F) {
    /* Sum: '<S56>/Sum' incorporates:
     *  DiscreteIntegrator: '<S46>/Integrator'
     *  Product: '<S51>/PProd Out'
     */
    rtb_Switch1 = (rtb_Sum1 * reg_FF_PI_pl_regr_stiff_B->Input11 +
                   reg_FF_PI_pl_regr_stiff_DW->Integrator_DSTATE_i) + rtb_Sum_d;

    /* Switch: '<S54>/Switch2' incorporates:
     *  Constant: '<S2>/max_sat'
     *  Constant: '<S2>/min_sat'
     *  RelationalOperator: '<S54>/LowerRelop1'
     *  RelationalOperator: '<S54>/UpperRelop'
     *  Sum: '<S2>/Sum3'
     *  Sum: '<S2>/Sum4'
     *  Switch: '<S54>/Switch'
     */
    if (rtb_Switch1 > 5.0 - reg_FF_PI_pl_regr_stiff_B->Input15) {
      rtb_Switch1 = 5.0 - reg_FF_PI_pl_regr_stiff_B->Input15;
    } else if (rtb_Switch1 < 0.0 - reg_FF_PI_pl_regr_stiff_B->Input15) {
      /* Switch: '<S54>/Switch' incorporates:
       *  Constant: '<S2>/min_sat'
       *  Sum: '<S2>/Sum4'
       */
      rtb_Switch1 = 0.0 - reg_FF_PI_pl_regr_stiff_B->Input15;
    }

    /* End of Switch: '<S54>/Switch2' */
  } else {
    rtb_Switch1 = 0.0;
  }

  /* End of Switch: '<Root>/Switch1' */

  /* MATLAB Function: '<S1>/MATLAB Function' incorporates:
   *  MultiPortSwitch: '<S1>/Multiport Switch1'
   */
  tmp[0] = AlphaY;
  tmp[1] = HTransform_tmp;
  tmp[2] = rtb_Blue_real;
  tmp[3] = rtb_Blue_ref;
  tmp[4] = tmp_1;
  tmp[5] = tmp_2;
  tmp[6] = reg_FF_PI_pl_regr_stiff_B->Input15;
  tmp[7] = 1.0F;
  rtb_Yellow_ref = 0.0F;
  for (i = 0; i < 8; i++) {
    rtb_Yellow_ref += (real32_T)rtb_MultiportSwitch1[6 * i] * tmp[i];
  }

  tmp[0] = AlphaY;
  tmp[1] = HTransform_tmp;
  tmp[2] = rtb_Blue_real;
  tmp[3] = rtb_Blue_ref;
  tmp[4] = tmp_1;
  tmp[5] = tmp_2;
  tmp[6] = reg_FF_PI_pl_regr_stiff_B->Input15;
  tmp[7] = 1.0F;
  rtb_Yellow_real = 0.0F;
  for (i = 0; i < 8; i++) {
    rtb_Yellow_real += (real32_T)rtb_MultiportSwitch1[6 * i + 1] * tmp[i];
  }

  tmp[0] = AlphaY;
  tmp[1] = HTransform_tmp;
  tmp[2] = rtb_Blue_real;
  tmp[3] = rtb_Blue_ref;
  tmp[4] = tmp_1;
  tmp[5] = tmp_2;
  tmp[6] = reg_FF_PI_pl_regr_stiff_B->Input15;
  tmp[7] = 1.0F;
  AlphaX = 0.0F;
  for (i = 0; i < 8; i++) {
    AlphaX += (real32_T)rtb_MultiportSwitch1[6 * i + 2] * tmp[i];
  }

  tmp[0] = AlphaY;
  tmp[1] = HTransform_tmp;
  tmp[2] = rtb_Blue_real;
  tmp[3] = rtb_Blue_ref;
  tmp[4] = tmp_1;
  tmp[5] = tmp_2;
  tmp[6] = reg_FF_PI_pl_regr_stiff_B->Input15;
  tmp[7] = 1.0F;
  rtb_Green_ref = 0.0F;
  for (i = 0; i < 8; i++) {
    rtb_Green_ref += (real32_T)rtb_MultiportSwitch1[6 * i + 3] * tmp[i];
  }

  tmp[0] = AlphaY;
  tmp[1] = HTransform_tmp;
  tmp[2] = rtb_Blue_real;
  tmp[3] = rtb_Blue_ref;
  tmp[4] = tmp_1;
  tmp[5] = tmp_2;
  tmp[6] = reg_FF_PI_pl_regr_stiff_B->Input15;
  tmp[7] = 1.0F;
  rtb_MultiportSwitch_1 = 0.0F;
  for (i = 0; i < 8; i++) {
    rtb_MultiportSwitch_1 += (real32_T)rtb_MultiportSwitch1[6 * i + 4] * tmp[i];
  }

  tmp[0] = AlphaY;
  tmp[1] = HTransform_tmp;
  tmp[2] = rtb_Blue_real;
  tmp[3] = rtb_Blue_ref;
  tmp[4] = tmp_1;
  tmp[5] = tmp_2;
  tmp[6] = reg_FF_PI_pl_regr_stiff_B->Input15;
  tmp[7] = 1.0F;
  AlphaY = 0.0F;
  for (i = 0; i < 8; i++) {
    AlphaY += (real32_T)rtb_MultiportSwitch1[6 * i + 5] * tmp[i];
  }

  rtb_MultiportSwitch_0[0] = rtb_Yellow_ref;
  rtb_MultiportSwitch_0[1] = rtb_Yellow_real;
  rtb_MultiportSwitch_0[2] = AlphaX;
  rtb_MultiportSwitch_0[3] = rtb_Green_ref;
  rtb_MultiportSwitch_0[4] = rtb_MultiportSwitch_1;
  rtb_MultiportSwitch_0[5] = AlphaY;
  tmp_0[0] = 1.0F;
  tmp_0[1] = reg_FF_PI_pl_regr_stiff_B->Input1;
  tmp_0[2] = reg_FF_PI_pl_regr_stiff_B->Input2;
  tmp_0[3] = rtb_MultiportSwitch_2;
  tmp_0[4] = rtb_MultiportSwitch_3;
  tmp_0[5] = rtb_MultiportSwitch_4;
  rtb_Yellow_ref = 0.0F;
  for (i = 0; i < 6; i++) {
    rtb_Yellow_ref += rtb_MultiportSwitch_0[i] * tmp_0[i];
  }

  /* Sum: '<Root>/Sum1' incorporates:
   *  MATLAB Function: '<S1>/MATLAB Function'
   */
  reg_FF_PI_pl_regr_stiff_B->Sum1 = (real32_T)(rtb_Switch1 + rtb_Yellow_ref);

  /* S-Function (bur_out): '<Root>/Output4' */
  inst->Green_tab = reg_FF_PI_pl_regr_stiff_B->Sum1;

  /* S-Function (bur_in): '<Root>/Input10' */
  reg_FF_PI_pl_regr_stiff_B->Input10 = inst->tlak3;

  /* S-Function (bur_in): '<Root>/Input12' */
  reg_FF_PI_pl_regr_stiff_B->Input12 = inst->I_parameter;

  /* S-Function (bur_in): '<Root>/Input8' */
  reg_FF_PI_pl_regr_stiff_B->Input8 = inst->tlak1;

  /* S-Function (bur_in): '<Root>/Input9' */
  reg_FF_PI_pl_regr_stiff_B->Input9 = inst->tlak2;

  /* Product: '<S43>/IProd Out' */
  rtb_Switch1 = rtb_Sum1 * reg_FF_PI_pl_regr_stiff_B->Input12;

  /* Product: '<S92>/IProd Out' */
  rtb_Sum2 *= reg_FF_PI_pl_regr_stiff_B->Input12;

  /* Product: '<S141>/IProd Out' */
  A2 *= reg_FF_PI_pl_regr_stiff_B->Input12;

  /* Update for DiscreteIntegrator: '<S144>/Integrator' */
  reg_FF_PI_pl_regr_stiff_DW->Integrator_DSTATE += 0.002 * A2;
  if (reg_FF_PI_pl_regr_stiff_B->Input5 > 0.0F) {
    reg_FF_PI_pl_regr_stiff_DW->Integrator_PrevResetState = 1;
  } else if (reg_FF_PI_pl_regr_stiff_B->Input5 < 0.0F) {
    reg_FF_PI_pl_regr_stiff_DW->Integrator_PrevResetState = -1;
  } else if (reg_FF_PI_pl_regr_stiff_B->Input5 == 0.0F) {
    reg_FF_PI_pl_regr_stiff_DW->Integrator_PrevResetState = 0;
  } else {
    reg_FF_PI_pl_regr_stiff_DW->Integrator_PrevResetState = 2;
  }

  /* End of Update for DiscreteIntegrator: '<S144>/Integrator' */

  /* Update for DiscreteIntegrator: '<S139>/Filter' */
  reg_FF_PI_pl_regr_stiff_DW->Filter_DSTATE += 0.002 * A1;
  if (reg_FF_PI_pl_regr_stiff_B->Input5 > 0.0F) {
    reg_FF_PI_pl_regr_stiff_DW->Filter_PrevResetState = 1;
  } else if (reg_FF_PI_pl_regr_stiff_B->Input5 < 0.0F) {
    reg_FF_PI_pl_regr_stiff_DW->Filter_PrevResetState = -1;
  } else if (reg_FF_PI_pl_regr_stiff_B->Input5 == 0.0F) {
    reg_FF_PI_pl_regr_stiff_DW->Filter_PrevResetState = 0;
  } else {
    reg_FF_PI_pl_regr_stiff_DW->Filter_PrevResetState = 2;
  }

  /* End of Update for DiscreteIntegrator: '<S139>/Filter' */

  /* Update for DiscreteIntegrator: '<S95>/Integrator' */
  reg_FF_PI_pl_regr_stiff_DW->Integrator_DSTATE_o += 0.002 * rtb_Sum2;
  if (reg_FF_PI_pl_regr_stiff_B->Input7 > 0.0F) {
    reg_FF_PI_pl_regr_stiff_DW->Integrator_PrevResetState_l = 1;
  } else if (reg_FF_PI_pl_regr_stiff_B->Input7 < 0.0F) {
    reg_FF_PI_pl_regr_stiff_DW->Integrator_PrevResetState_l = -1;
  } else if (reg_FF_PI_pl_regr_stiff_B->Input7 == 0.0F) {
    reg_FF_PI_pl_regr_stiff_DW->Integrator_PrevResetState_l = 0;
  } else {
    reg_FF_PI_pl_regr_stiff_DW->Integrator_PrevResetState_l = 2;
  }

  /* End of Update for DiscreteIntegrator: '<S95>/Integrator' */

  /* Update for DiscreteIntegrator: '<S90>/Filter' */
  reg_FF_PI_pl_regr_stiff_DW->Filter_DSTATE_f += 0.002 * A3;
  if (reg_FF_PI_pl_regr_stiff_B->Input7 > 0.0F) {
    reg_FF_PI_pl_regr_stiff_DW->Filter_PrevResetState_e = 1;
  } else if (reg_FF_PI_pl_regr_stiff_B->Input7 < 0.0F) {
    reg_FF_PI_pl_regr_stiff_DW->Filter_PrevResetState_e = -1;
  } else if (reg_FF_PI_pl_regr_stiff_B->Input7 == 0.0F) {
    reg_FF_PI_pl_regr_stiff_DW->Filter_PrevResetState_e = 0;
  } else {
    reg_FF_PI_pl_regr_stiff_DW->Filter_PrevResetState_e = 2;
  }

  /* End of Update for DiscreteIntegrator: '<S90>/Filter' */

  /* Update for DiscreteIntegrator: '<S46>/Integrator' */
  reg_FF_PI_pl_regr_stiff_DW->Integrator_DSTATE_i += 0.002 * rtb_Switch1;
  if (reg_FF_PI_pl_regr_stiff_B->Input6 > 0.0F) {
    reg_FF_PI_pl_regr_stiff_DW->Integrator_PrevResetState_e = 1;
  } else if (reg_FF_PI_pl_regr_stiff_B->Input6 < 0.0F) {
    reg_FF_PI_pl_regr_stiff_DW->Integrator_PrevResetState_e = -1;
  } else if (reg_FF_PI_pl_regr_stiff_B->Input6 == 0.0F) {
    reg_FF_PI_pl_regr_stiff_DW->Integrator_PrevResetState_e = 0;
  } else {
    reg_FF_PI_pl_regr_stiff_DW->Integrator_PrevResetState_e = 2;
  }

  /* End of Update for DiscreteIntegrator: '<S46>/Integrator' */

  /* Update for DiscreteIntegrator: '<S41>/Filter' */
  reg_FF_PI_pl_regr_stiff_DW->Filter_DSTATE_a += 0.002 * rtb_Sum_d;
  if (reg_FF_PI_pl_regr_stiff_B->Input6 > 0.0F) {
    reg_FF_PI_pl_regr_stiff_DW->Filter_PrevResetState_h = 1;
  } else if (reg_FF_PI_pl_regr_stiff_B->Input6 < 0.0F) {
    reg_FF_PI_pl_regr_stiff_DW->Filter_PrevResetState_h = -1;
  } else if (reg_FF_PI_pl_regr_stiff_B->Input6 == 0.0F) {
    reg_FF_PI_pl_regr_stiff_DW->Filter_PrevResetState_h = 0;
  } else {
    reg_FF_PI_pl_regr_stiff_DW->Filter_PrevResetState_h = 2;
  }

  /* End of Update for DiscreteIntegrator: '<S41>/Filter' */
}

/* Model initialize function */
void reg_FF_PI_pl_regr_stiff_initialize(RT_MODEL_reg_FF_PI_pl_regr_st_T *const
  reg_FF_PI_pl_regr_stiff_M, struct FF_PID_r_t* inst)
{
  DW_reg_FF_PI_pl_regr_stiff_T *reg_FF_PI_pl_regr_stiff_DW =
    reg_FF_PI_pl_regr_stiff_M->dwork;

  /* InitializeConditions for DiscreteIntegrator: '<S144>/Integrator' */
  reg_FF_PI_pl_regr_stiff_DW->Integrator_DSTATE = 0.0;
  reg_FF_PI_pl_regr_stiff_DW->Integrator_PrevResetState = 2;

  /* InitializeConditions for DiscreteIntegrator: '<S139>/Filter' */
  reg_FF_PI_pl_regr_stiff_DW->Filter_DSTATE = 0.0;
  reg_FF_PI_pl_regr_stiff_DW->Filter_PrevResetState = 2;

  /* InitializeConditions for DiscreteIntegrator: '<S95>/Integrator' */
  reg_FF_PI_pl_regr_stiff_DW->Integrator_DSTATE_o = 0.0;
  reg_FF_PI_pl_regr_stiff_DW->Integrator_PrevResetState_l = 2;

  /* InitializeConditions for DiscreteIntegrator: '<S90>/Filter' */
  reg_FF_PI_pl_regr_stiff_DW->Filter_DSTATE_f = 0.0;
  reg_FF_PI_pl_regr_stiff_DW->Filter_PrevResetState_e = 2;

  /* InitializeConditions for DiscreteIntegrator: '<S46>/Integrator' */
  reg_FF_PI_pl_regr_stiff_DW->Integrator_DSTATE_i = 0.0;
  reg_FF_PI_pl_regr_stiff_DW->Integrator_PrevResetState_e = 2;

  /* InitializeConditions for DiscreteIntegrator: '<S41>/Filter' */
  reg_FF_PI_pl_regr_stiff_DW->Filter_DSTATE_a = 0.0;
  reg_FF_PI_pl_regr_stiff_DW->Filter_PrevResetState_h = 2;
}

/* Model terminate function */
void reg_FF_PI_pl_regr_stiff_terminate(RT_MODEL_reg_FF_PI_pl_regr_st_T
  * reg_FF_PI_pl_regr_stiff_M, struct FF_PID_r_t* inst)
{}

/* Model data allocation function */
void reg_FF_PI_pl_regr_stiff_initializeMemory(RT_MODEL_reg_FF_PI_pl_regr_st_T* const reg_FF_PI_pl_regr_stiff_M, struct FF_PID_r_t * inst)
{  /* states (dwork) */
  {
  }

  {
    B_reg_FF_PI_pl_regr_stiff_T *reg_FF_PI_pl_regr_stiff_B =
      reg_FF_PI_pl_regr_stiff_M->blockIO;
    DW_reg_FF_PI_pl_regr_stiff_T *reg_FF_PI_pl_regr_stiff_DW =
      reg_FF_PI_pl_regr_stiff_M->dwork;

    /* block I/O */
    {
      reg_FF_PI_pl_regr_stiff_B->Input15 = 0.0F;
      reg_FF_PI_pl_regr_stiff_B->Input1 = 0.0F;
      reg_FF_PI_pl_regr_stiff_B->Input2 = 0.0F;
      reg_FF_PI_pl_regr_stiff_B->Input3 = 0.0F;
      reg_FF_PI_pl_regr_stiff_B->Input4 = 0.0F;
      reg_FF_PI_pl_regr_stiff_B->Input16 = 0.0F;
      reg_FF_PI_pl_regr_stiff_B->Input11 = 0.0F;
      reg_FF_PI_pl_regr_stiff_B->Input5 = 0.0F;
      reg_FF_PI_pl_regr_stiff_B->Input13 = 0.0F;
      reg_FF_PI_pl_regr_stiff_B->Input14 = 0.0F;
      reg_FF_PI_pl_regr_stiff_B->Input17 = 0.0F;
      reg_FF_PI_pl_regr_stiff_B->Sum = 0.0F;
      reg_FF_PI_pl_regr_stiff_B->Input7 = 0.0F;
      reg_FF_PI_pl_regr_stiff_B->Sum2 = 0.0F;
      reg_FF_PI_pl_regr_stiff_B->Input6 = 0.0F;
      reg_FF_PI_pl_regr_stiff_B->Sum1 = 0.0F;
      reg_FF_PI_pl_regr_stiff_B->Input10 = 0.0F;
      reg_FF_PI_pl_regr_stiff_B->Input12 = 0.0F;
      reg_FF_PI_pl_regr_stiff_B->Input8 = 0.0F;
      reg_FF_PI_pl_regr_stiff_B->Input9 = 0.0F;
    }

    /* states (dwork) */
    (void) memset((void *)reg_FF_PI_pl_regr_stiff_DW, 0,
                  sizeof(DW_reg_FF_PI_pl_regr_stiff_T));
    reg_FF_PI_pl_regr_stiff_DW->Integrator_DSTATE = 0.0;
    reg_FF_PI_pl_regr_stiff_DW->Filter_DSTATE = 0.0;
    reg_FF_PI_pl_regr_stiff_DW->Integrator_DSTATE_o = 0.0;
    reg_FF_PI_pl_regr_stiff_DW->Filter_DSTATE_f = 0.0;
    reg_FF_PI_pl_regr_stiff_DW->Integrator_DSTATE_i = 0.0;
    reg_FF_PI_pl_regr_stiff_DW->Filter_DSTATE_a = 0.0;
  }

}
```
